REGION Network 4: Functional Test Station 6
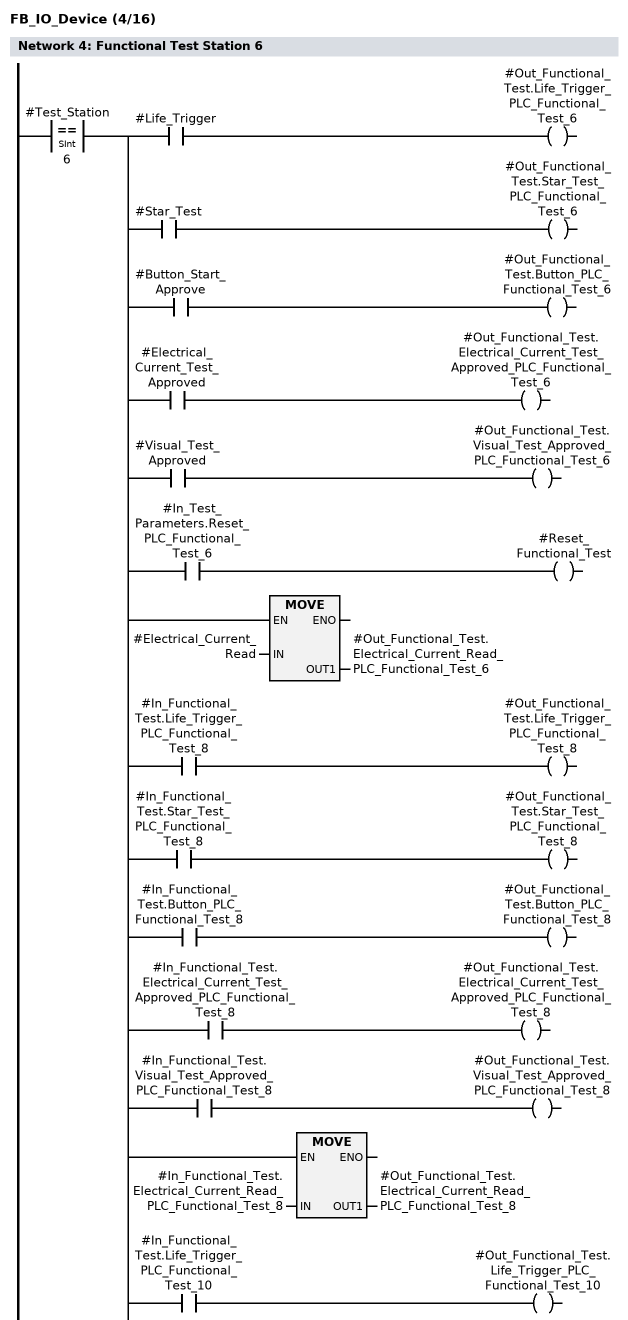
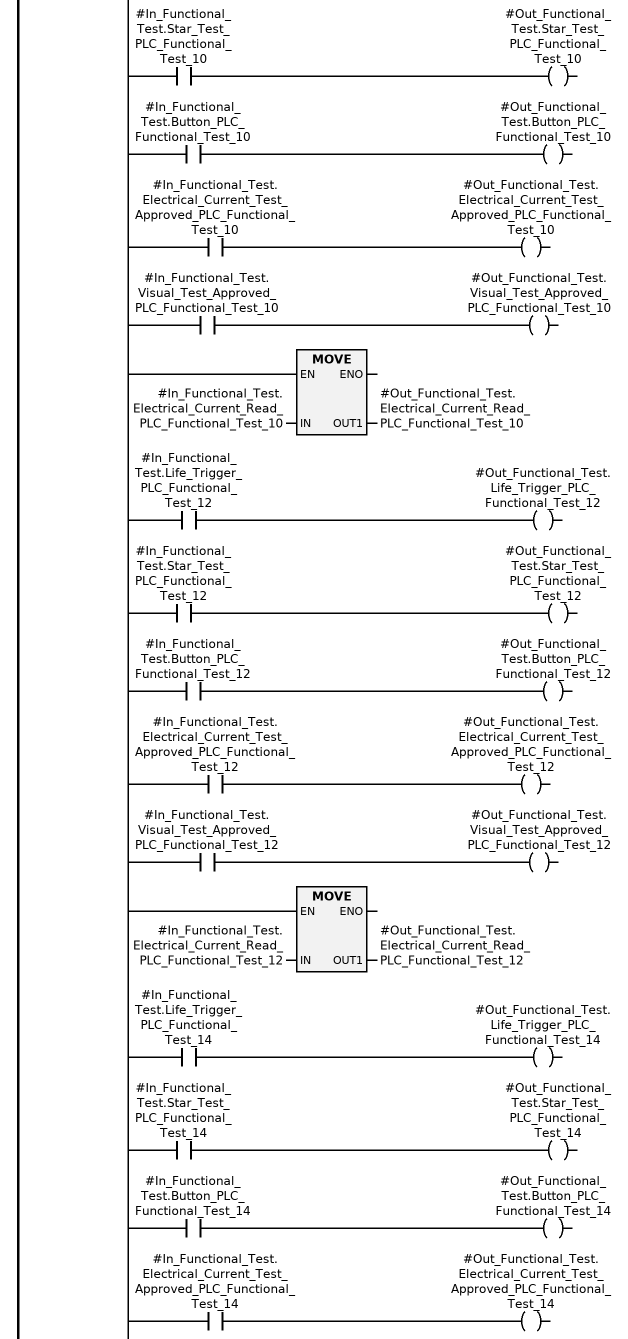
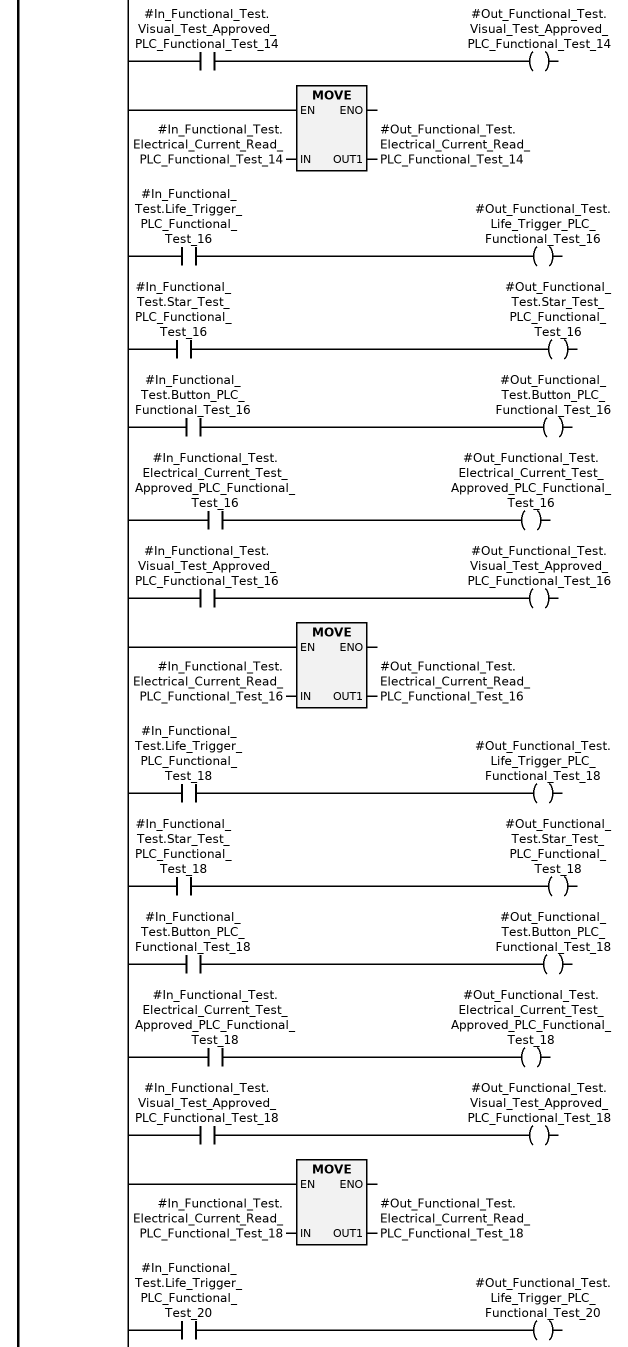
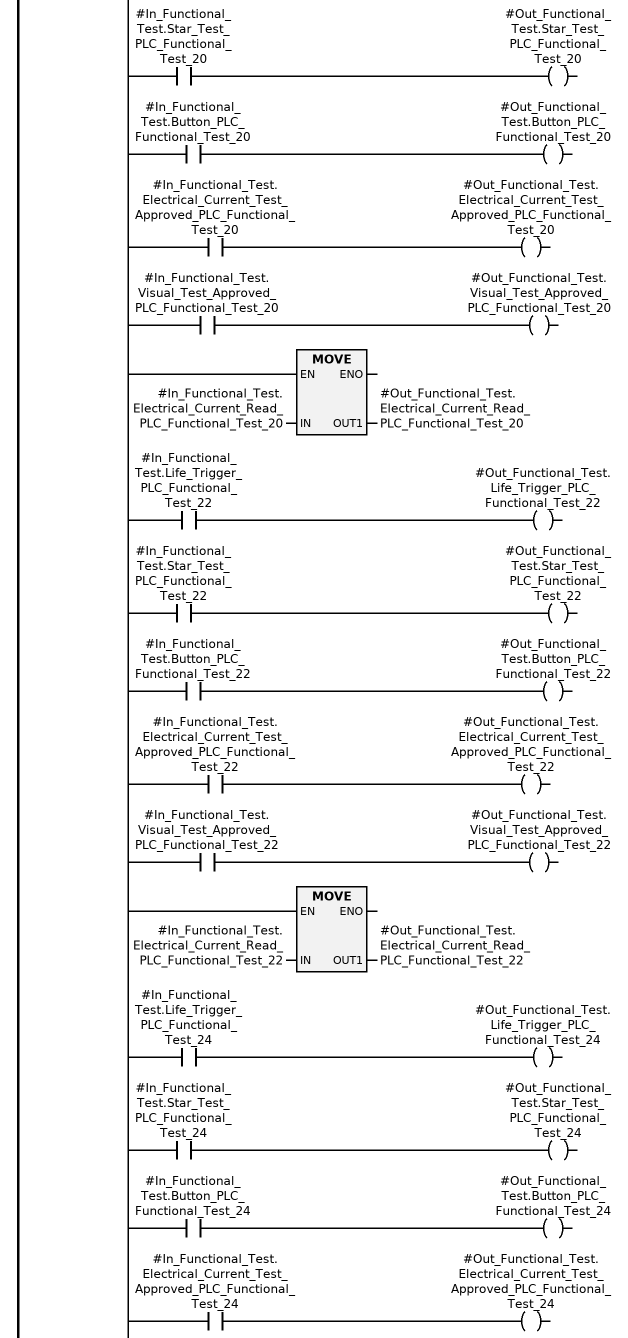
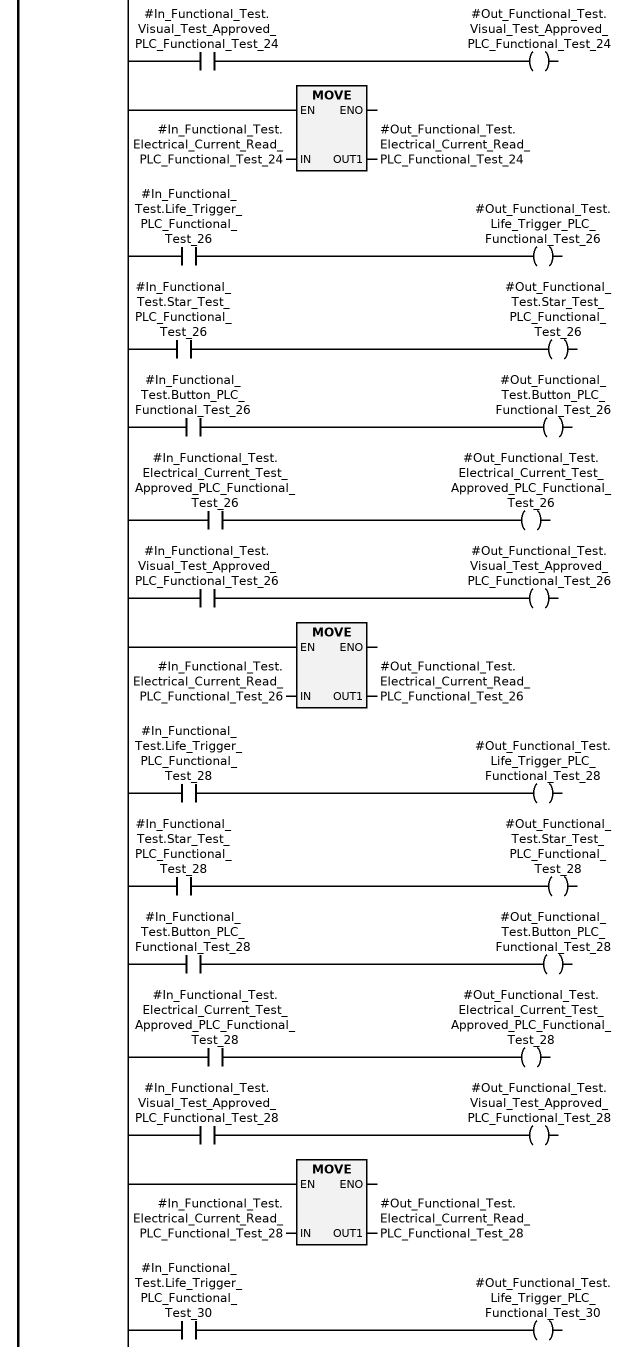
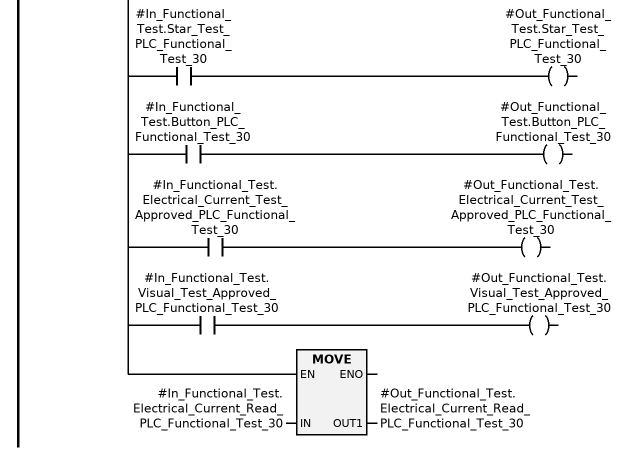
   RUNG wire#powerrail
      { S7_Templates := "SrcType := SInt" } EQ_Contact(in1 := #Test_Station, in2 := 6)
      wire#w1
      Contact( #Life_Trigger )
      Coil( #Out_Functional_Test.Life_Trigger_PLC_Functional_Test_6 )
   END_RUNG
   RUNG wire#w1
      Contact( #Star_Test )
      Coil( #Out_Functional_Test.Star_Test_PLC_Functional_Test_6 )
   END_RUNG
   RUNG wire#w1
      Contact( #Button_Start_Approve )
      Coil( #Out_Functional_Test.Button_PLC_Functional_Test_6 )
   END_RUNG
   RUNG wire#w1
      Contact( #Electrical_Current_Test_Approved )
      Coil( #Out_Functional_Test.Electrical_Current_Test_Approved_PLC_Functional_Test_6 )
   END_RUNG
   RUNG wire#w1
      Contact( #Visual_Test_Approved )
      Coil( #Out_Functional_Test.Visual_Test_Approved_PLC_Functional_Test_6 )
   END_RUNG
   RUNG wire#w1
      Contact( #In_Test_Parameters.Reset_PLC_Functional_Test_6 )
      Coil( #Reset_Functional_Test )
   END_RUNG
   RUNG wire#w1
      Move(in := #Electrical_Current_Read, out1 => #Out_Functional_Test.Electrical_Current_Read_PLC_Functional_Test_6)
   END_RUNG
   RUNG wire#w1
      Contact( #In_Functional_Test.Life_Trigger_PLC_Functional_Test_8 )
      Coil( #Out_Functional_Test.Life_Trigger_PLC_Functional_Test_8 )
   END_RUNG
   RUNG wire#w1
      Contact( #In_Functional_Test.Star_Test_PLC_Functional_Test_8 )
      Coil( #Out_Functional_Test.Star_Test_PLC_Functional_Test_8 )
   END_RUNG
   RUNG wire#w1
      Contact( #In_Functional_Test.Button_PLC_Functional_Test_8 )
      Coil( #Out_Functional_Test.Button_PLC_Functional_Test_8 )
   END_RUNG
   RUNG wire#w1
      Contact( #In_Functional_Test.Electrical_Current_Test_Approved_PLC_Functional_Test_8 )
      Coil( #Out_Functional_Test.Electrical_Current_Test_Approved_PLC_Functional_Test_8 )
   END_RUNG
   RUNG wire#w1
      Contact( #In_Functional_Test.Visual_Test_Approved_PLC_Functional_Test_8 )
      Coil( #Out_Functional_Test.Visual_Test_Approved_PLC_Functional_Test_8 )
   END_RUNG
   RUNG wire#w1
      Move(in := #In_Functional_Test.Electrical_Current_Read_PLC_Functional_Test_8, out1 => #Out_Functional_Test.Electrical_Current_Read_PLC_Functional_Test_8)
   END_RUNG
   RUNG wire#w1
      Contact( #In_Functional_Test.Life_Trigger_PLC_Functional_Test_10 )
      Coil( #Out_Functional_Test.Life_Trigger_PLC_Functional_Test_10 )
   END_RUNG
   RUNG wire#w1
      Contact( #In_Functional_Test.Star_Test_PLC_Functional_Test_10 )
      Coil( #Out_Functional_Test.Star_Test_PLC_Functional_Test_10 )
   END_RUNG
   RUNG wire#w1
      Contact( #In_Functional_Test.Button_PLC_Functional_Test_10 )
      Coil( #Out_Functional_Test.Button_PLC_Functional_Test_10 )
   END_RUNG
   RUNG wire#w1
      Contact( #In_Functional_Test.Electrical_Current_Test_Approved_PLC_Functional_Test_10 )
      Coil( #Out_Functional_Test.Electrical_Current_Test_Approved_PLC_Functional_Test_10 )
   END_RUNG
   RUNG wire#w1
      Contact( #In_Functional_Test.Visual_Test_Approved_PLC_Functional_Test_10 )
      Coil( #Out_Functional_Test.Visual_Test_Approved_PLC_Functional_Test_10 )
   END_RUNG
   RUNG wire#w1
      Move(in := #In_Functional_Test.Electrical_Current_Read_PLC_Functional_Test_10, out1 => #Out_Functional_Test.Electrical_Current_Read_PLC_Functional_Test_10)
   END_RUNG
   RUNG wire#w1
      Contact( #In_Functional_Test.Life_Trigger_PLC_Functional_Test_12 )
      Coil( #Out_Functional_Test.Life_Trigger_PLC_Functional_Test_12 )
   END_RUNG
   RUNG wire#w1
      Contact( #In_Functional_Test.Star_Test_PLC_Functional_Test_12 )
      Coil( #Out_Functional_Test.Star_Test_PLC_Functional_Test_12 )
   END_RUNG
   RUNG wire#w1
      Contact( #In_Functional_Test.Button_PLC_Functional_Test_12 )
      Coil( #Out_Functional_Test.Button_PLC_Functional_Test_12 )
   END_RUNG
   RUNG wire#w1
      Contact( #In_Functional_Test.Electrical_Current_Test_Approved_PLC_Functional_Test_12 )
      Coil( #Out_Functional_Test.Electrical_Current_Test_Approved_PLC_Functional_Test_12 )
   END_RUNG
   RUNG wire#w1
      Contact( #In_Functional_Test.Visual_Test_Approved_PLC_Functional_Test_12 )
      Coil( #Out_Functional_Test.Visual_Test_Approved_PLC_Functional_Test_12 )
   END_RUNG
   RUNG wire#w1
      Move(in := #In_Functional_Test.Electrical_Current_Read_PLC_Functional_Test_12, out1 => #Out_Functional_Test.Electrical_Current_Read_PLC_Functional_Test_12)
   END_RUNG
   RUNG wire#w1
      Contact( #In_Functional_Test.Life_Trigger_PLC_Functional_Test_14 )
      Coil( #Out_Functional_Test.Life_Trigger_PLC_Functional_Test_14 )
   END_RUNG
   RUNG wire#w1
      Contact( #In_Functional_Test.Star_Test_PLC_Functional_Test_14 )
      Coil( #Out_Functional_Test.Star_Test_PLC_Functional_Test_14 )
   END_RUNG
   RUNG wire#w1
      Contact( #In_Functional_Test.Button_PLC_Functional_Test_14 )
      Coil( #Out_Functional_Test.Button_PLC_Functional_Test_14 )
   END_RUNG
   RUNG wire#w1
      Contact( #In_Functional_Test.Electrical_Current_Test_Approved_PLC_Functional_Test_14 )
      Coil( #Out_Functional_Test.Electrical_Current_Test_Approved_PLC_Functional_Test_14 )
   END_RUNG
   RUNG wire#w1
      Contact( #In_Functional_Test.Visual_Test_Approved_PLC_Functional_Test_14 )
      Coil( #Out_Functional_Test.Visual_Test_Approved_PLC_Functional_Test_14 )
   END_RUNG
   RUNG wire#w1
      Move(in := #In_Functional_Test.Electrical_Current_Read_PLC_Functional_Test_14, out1 => #Out_Functional_Test.Electrical_Current_Read_PLC_Functional_Test_14)
   END_RUNG
   RUNG wire#w1
      Contact( #In_Functional_Test.Life_Trigger_PLC_Functional_Test_16 )
      Coil( #Out_Functional_Test.Life_Trigger_PLC_Functional_Test_16 )
   END_RUNG
   RUNG wire#w1
      Contact( #In_Functional_Test.Star_Test_PLC_Functional_Test_16 )
      Coil( #Out_Functional_Test.Star_Test_PLC_Functional_Test_16 )
   END_RUNG
   RUNG wire#w1
      Contact( #In_Functional_Test.Button_PLC_Functional_Test_16 )
      Coil( #Out_Functional_Test.Button_PLC_Functional_Test_16 )
   END_RUNG
   RUNG wire#w1
      Contact( #In_Functional_Test.Electrical_Current_Test_Approved_PLC_Functional_Test_16 )
      Coil( #Out_Functional_Test.Electrical_Current_Test_Approved_PLC_Functional_Test_16 )
   END_RUNG
   RUNG wire#w1
      Contact( #In_Functional_Test.Visual_Test_Approved_PLC_Functional_Test_16 )
      Coil( #Out_Functional_Test.Visual_Test_Approved_PLC_Functional_Test_16 )
   END_RUNG
   RUNG wire#w1
      Move(in := #In_Functional_Test.Electrical_Current_Read_PLC_Functional_Test_16, out1 => #Out_Functional_Test.Electrical_Current_Read_PLC_Functional_Test_16)
   END_RUNG
   RUNG wire#w1
      Contact( #In_Functional_Test.Life_Trigger_PLC_Functional_Test_18 )
      Coil( #Out_Functional_Test.Life_Trigger_PLC_Functional_Test_18 )
   END_RUNG
   RUNG wire#w1
      Contact( #In_Functional_Test.Star_Test_PLC_Functional_Test_18 )
      Coil( #Out_Functional_Test.Star_Test_PLC_Functional_Test_18 )
   END_RUNG
   RUNG wire#w1
      Contact( #In_Functional_Test.Button_PLC_Functional_Test_18 )
      Coil( #Out_Functional_Test.Button_PLC_Functional_Test_18 )
   END_RUNG
   RUNG wire#w1
      Contact( #In_Functional_Test.Electrical_Current_Test_Approved_PLC_Functional_Test_18 )
      Coil( #Out_Functional_Test.Electrical_Current_Test_Approved_PLC_Functional_Test_18 )
   END_RUNG
   RUNG wire#w1
      Contact( #In_Functional_Test.Visual_Test_Approved_PLC_Functional_Test_18 )
      Coil( #Out_Functional_Test.Visual_Test_Approved_PLC_Functional_Test_18 )
   END_RUNG
   RUNG wire#w1
      Move(in := #In_Functional_Test.Electrical_Current_Read_PLC_Functional_Test_18, out1 => #Out_Functional_Test.Electrical_Current_Read_PLC_Functional_Test_18)
   END_RUNG
   RUNG wire#w1
      Contact( #In_Functional_Test.Life_Trigger_PLC_Functional_Test_20 )
      Coil( #Out_Functional_Test.Life_Trigger_PLC_Functional_Test_20 )
   END_RUNG
   RUNG wire#w1
      Contact( #In_Functional_Test.Star_Test_PLC_Functional_Test_20 )
      Coil( #Out_Functional_Test.Star_Test_PLC_Functional_Test_20 )
   END_RUNG
   RUNG wire#w1
      Contact( #In_Functional_Test.Button_PLC_Functional_Test_20 )
      Coil( #Out_Functional_Test.Button_PLC_Functional_Test_20 )
   END_RUNG
   RUNG wire#w1
      Contact( #In_Functional_Test.Electrical_Current_Test_Approved_PLC_Functional_Test_20 )
      Coil( #Out_Functional_Test.Electrical_Current_Test_Approved_PLC_Functional_Test_20 )
   END_RUNG
   RUNG wire#w1
      Contact( #In_Functional_Test.Visual_Test_Approved_PLC_Functional_Test_20 )
      Coil( #Out_Functional_Test.Visual_Test_Approved_PLC_Functional_Test_20 )
   END_RUNG
   RUNG wire#w1
      Move(in := #In_Functional_Test.Electrical_Current_Read_PLC_Functional_Test_20, out1 => #Out_Functional_Test.Electrical_Current_Read_PLC_Functional_Test_20)
   END_RUNG
   RUNG wire#w1
      Contact( #In_Functional_Test.Life_Trigger_PLC_Functional_Test_22 )
      Coil( #Out_Functional_Test.Life_Trigger_PLC_Functional_Test_22 )
   END_RUNG
   RUNG wire#w1
      Contact( #In_Functional_Test.Star_Test_PLC_Functional_Test_22 )
      Coil( #Out_Functional_Test.Star_Test_PLC_Functional_Test_22 )
   END_RUNG
   RUNG wire#w1
      Contact( #In_Functional_Test.Button_PLC_Functional_Test_22 )
      Coil( #Out_Functional_Test.Button_PLC_Functional_Test_22 )
   END_RUNG
   RUNG wire#w1
      Contact( #In_Functional_Test.Electrical_Current_Test_Approved_PLC_Functional_Test_22 )
      Coil( #Out_Functional_Test.Electrical_Current_Test_Approved_PLC_Functional_Test_22 )
   END_RUNG
   RUNG wire#w1
      Contact( #In_Functional_Test.Visual_Test_Approved_PLC_Functional_Test_22 )
      Coil( #Out_Functional_Test.Visual_Test_Approved_PLC_Functional_Test_22 )
   END_RUNG
   RUNG wire#w1
      Move(in := #In_Functional_Test.Electrical_Current_Read_PLC_Functional_Test_22, out1 => #Out_Functional_Test.Electrical_Current_Read_PLC_Functional_Test_22)
   END_RUNG
   RUNG wire#w1
      Contact( #In_Functional_Test.Life_Trigger_PLC_Functional_Test_24 )
      Coil( #Out_Functional_Test.Life_Trigger_PLC_Functional_Test_24 )
   END_RUNG
   RUNG wire#w1
      Contact( #In_Functional_Test.Star_Test_PLC_Functional_Test_24 )
      Coil( #Out_Functional_Test.Star_Test_PLC_Functional_Test_24 )
   END_RUNG
   RUNG wire#w1
      Contact( #In_Functional_Test.Button_PLC_Functional_Test_24 )
      Coil( #Out_Functional_Test.Button_PLC_Functional_Test_24 )
   END_RUNG
   RUNG wire#w1
      Contact( #In_Functional_Test.Electrical_Current_Test_Approved_PLC_Functional_Test_24 )
      Coil( #Out_Functional_Test.Electrical_Current_Test_Approved_PLC_Functional_Test_24 )
   END_RUNG
   RUNG wire#w1
      Contact( #In_Functional_Test.Visual_Test_Approved_PLC_Functional_Test_24 )
      Coil( #Out_Functional_Test.Visual_Test_Approved_PLC_Functional_Test_24 )
   END_RUNG
   RUNG wire#w1
      Move(in := #In_Functional_Test.Electrical_Current_Read_PLC_Functional_Test_24, out1 => #Out_Functional_Test.Electrical_Current_Read_PLC_Functional_Test_24)
   END_RUNG
   RUNG wire#w1
      Contact( #In_Functional_Test.Life_Trigger_PLC_Functional_Test_26 )
      Coil( #Out_Functional_Test.Life_Trigger_PLC_Functional_Test_26 )
   END_RUNG
   RUNG wire#w1
      Contact( #In_Functional_Test.Star_Test_PLC_Functional_Test_26 )
      Coil( #Out_Functional_Test.Star_Test_PLC_Functional_Test_26 )
   END_RUNG
   RUNG wire#w1
      Contact( #In_Functional_Test.Button_PLC_Functional_Test_26 )
      Coil( #Out_Functional_Test.Button_PLC_Functional_Test_26 )
   END_RUNG
   RUNG wire#w1
      Contact( #In_Functional_Test.Electrical_Current_Test_Approved_PLC_Functional_Test_26 )
      Coil( #Out_Functional_Test.Electrical_Current_Test_Approved_PLC_Functional_Test_26 )
   END_RUNG
   RUNG wire#w1
      Contact( #In_Functional_Test.Visual_Test_Approved_PLC_Functional_Test_26 )
      Coil( #Out_Functional_Test.Visual_Test_Approved_PLC_Functional_Test_26 )
   END_RUNG
   RUNG wire#w1
      Move(in := #In_Functional_Test.Electrical_Current_Read_PLC_Functional_Test_26, out1 => #Out_Functional_Test.Electrical_Current_Read_PLC_Functional_Test_26)
   END_RUNG
   RUNG wire#w1
      Contact( #In_Functional_Test.Life_Trigger_PLC_Functional_Test_28 )
      Coil( #Out_Functional_Test.Life_Trigger_PLC_Functional_Test_28 )
   END_RUNG
   RUNG wire#w1
      Contact( #In_Functional_Test.Star_Test_PLC_Functional_Test_28 )
      Coil( #Out_Functional_Test.Star_Test_PLC_Functional_Test_28 )
   END_RUNG
   RUNG wire#w1
      Contact( #In_Functional_Test.Button_PLC_Functional_Test_28 )
      Coil( #Out_Functional_Test.Button_PLC_Functional_Test_28 )
   END_RUNG
   RUNG wire#w1
      Contact( #In_Functional_Test.Electrical_Current_Test_Approved_PLC_Functional_Test_28 )
      Coil( #Out_Functional_Test.Electrical_Current_Test_Approved_PLC_Functional_Test_28 )
   END_RUNG
   RUNG wire#w1
      Contact( #In_Functional_Test.Visual_Test_Approved_PLC_Functional_Test_28 )
      Coil( #Out_Functional_Test.Visual_Test_Approved_PLC_Functional_Test_28 )
   END_RUNG
   RUNG wire#w1
      Move(in := #In_Functional_Test.Electrical_Current_Read_PLC_Functional_Test_28, out1 => #Out_Functional_Test.Electrical_Current_Read_PLC_Functional_Test_28)
   END_RUNG
   RUNG wire#w1
      Contact( #In_Functional_Test.Life_Trigger_PLC_Functional_Test_30 )
      Coil( #Out_Functional_Test.Life_Trigger_PLC_Functional_Test_30 )
   END_RUNG
   RUNG wire#w1
      Contact( #In_Functional_Test.Star_Test_PLC_Functional_Test_30 )
      Coil( #Out_Functional_Test.Star_Test_PLC_Functional_Test_30 )
   END_RUNG
   RUNG wire#w1
      Contact( #In_Functional_Test.Button_PLC_Functional_Test_30 )
      Coil( #Out_Functional_Test.Button_PLC_Functional_Test_30 )
   END_RUNG
   RUNG wire#w1
      Contact( #In_Functional_Test.Electrical_Current_Test_Approved_PLC_Functional_Test_30 )
      Coil( #Out_Functional_Test.Electrical_Current_Test_Approved_PLC_Functional_Test_30 )
   END_RUNG
   RUNG wire#w1
      Contact( #In_Functional_Test.Visual_Test_Approved_PLC_Functional_Test_30 )
      Coil( #Out_Functional_Test.Visual_Test_Approved_PLC_Functional_Test_30 )
   END_RUNG
   RUNG wire#w1
      Move(in := #In_Functional_Test.Electrical_Current_Read_PLC_Functional_Test_30, out1 => #Out_Functional_Test.Electrical_Current_Read_PLC_Functional_Test_30)
   END_RUNG
   // the same network as SCL:
   #_w1 := #Test_Station = 6;
   #Out_Functional_Test.Life_Trigger_PLC_Functional_Test_6 := #_w1 AND #Life_Trigger;
   #Out_Functional_Test.Star_Test_PLC_Functional_Test_6 := #_w1 AND #Star_Test;
   #Out_Functional_Test.Button_PLC_Functional_Test_6 := #_w1 AND #Button_Start_Approve;
   #Out_Functional_Test.Electrical_Current_Test_Approved_PLC_Functional_Test_6 := #_w1 AND #Electrical_Current_Test_Approved;
   #Out_Functional_Test.Visual_Test_Approved_PLC_Functional_Test_6 := #_w1 AND #Visual_Test_Approved;
   #Reset_Functional_Test := #_w1 AND #In_Test_Parameters.Reset_PLC_Functional_Test_6;
   IF #_w1 THEN
       #Out_Functional_Test.Electrical_Current_Read_PLC_Functional_Test_6 := #Electrical_Current_Read;
   END_IF;
   #Out_Functional_Test.Life_Trigger_PLC_Functional_Test_8 := #_w1 AND #In_Functional_Test.Life_Trigger_PLC_Functional_Test_8;
   #Out_Functional_Test.Star_Test_PLC_Functional_Test_8 := #_w1 AND #In_Functional_Test.Star_Test_PLC_Functional_Test_8;
   #Out_Functional_Test.Button_PLC_Functional_Test_8 := #_w1 AND #In_Functional_Test.Button_PLC_Functional_Test_8;
   #Out_Functional_Test.Electrical_Current_Test_Approved_PLC_Functional_Test_8 := #_w1 AND #In_Functional_Test.Electrical_Current_Test_Approved_PLC_Functional_Test_8;
   #Out_Functional_Test.Visual_Test_Approved_PLC_Functional_Test_8 := #_w1 AND #In_Functional_Test.Visual_Test_Approved_PLC_Functional_Test_8;
   IF #_w1 THEN
       #Out_Functional_Test.Electrical_Current_Read_PLC_Functional_Test_8 := #In_Functional_Test.Electrical_Current_Read_PLC_Functional_Test_8;
   END_IF;
   #Out_Functional_Test.Life_Trigger_PLC_Functional_Test_10 := #_w1 AND #In_Functional_Test.Life_Trigger_PLC_Functional_Test_10;
   #Out_Functional_Test.Star_Test_PLC_Functional_Test_10 := #_w1 AND #In_Functional_Test.Star_Test_PLC_Functional_Test_10;
   #Out_Functional_Test.Button_PLC_Functional_Test_10 := #_w1 AND #In_Functional_Test.Button_PLC_Functional_Test_10;
   #Out_Functional_Test.Electrical_Current_Test_Approved_PLC_Functional_Test_10 := #_w1 AND #In_Functional_Test.Electrical_Current_Test_Approved_PLC_Functional_Test_10;
   #Out_Functional_Test.Visual_Test_Approved_PLC_Functional_Test_10 := #_w1 AND #In_Functional_Test.Visual_Test_Approved_PLC_Functional_Test_10;
   IF #_w1 THEN
       #Out_Functional_Test.Electrical_Current_Read_PLC_Functional_Test_10 := #In_Functional_Test.Electrical_Current_Read_PLC_Functional_Test_10;
   END_IF;
   #Out_Functional_Test.Life_Trigger_PLC_Functional_Test_12 := #_w1 AND #In_Functional_Test.Life_Trigger_PLC_Functional_Test_12;
   #Out_Functional_Test.Star_Test_PLC_Functional_Test_12 := #_w1 AND #In_Functional_Test.Star_Test_PLC_Functional_Test_12;
   #Out_Functional_Test.Button_PLC_Functional_Test_12 := #_w1 AND #In_Functional_Test.Button_PLC_Functional_Test_12;
   #Out_Functional_Test.Electrical_Current_Test_Approved_PLC_Functional_Test_12 := #_w1 AND #In_Functional_Test.Electrical_Current_Test_Approved_PLC_Functional_Test_12;
   #Out_Functional_Test.Visual_Test_Approved_PLC_Functional_Test_12 := #_w1 AND #In_Functional_Test.Visual_Test_Approved_PLC_Functional_Test_12;
   IF #_w1 THEN
       #Out_Functional_Test.Electrical_Current_Read_PLC_Functional_Test_12 := #In_Functional_Test.Electrical_Current_Read_PLC_Functional_Test_12;
   END_IF;
   #Out_Functional_Test.Life_Trigger_PLC_Functional_Test_14 := #_w1 AND #In_Functional_Test.Life_Trigger_PLC_Functional_Test_14;
   #Out_Functional_Test.Star_Test_PLC_Functional_Test_14 := #_w1 AND #In_Functional_Test.Star_Test_PLC_Functional_Test_14;
   #Out_Functional_Test.Button_PLC_Functional_Test_14 := #_w1 AND #In_Functional_Test.Button_PLC_Functional_Test_14;
   #Out_Functional_Test.Electrical_Current_Test_Approved_PLC_Functional_Test_14 := #_w1 AND #In_Functional_Test.Electrical_Current_Test_Approved_PLC_Functional_Test_14;
   #Out_Functional_Test.Visual_Test_Approved_PLC_Functional_Test_14 := #_w1 AND #In_Functional_Test.Visual_Test_Approved_PLC_Functional_Test_14;
   IF #_w1 THEN
       #Out_Functional_Test.Electrical_Current_Read_PLC_Functional_Test_14 := #In_Functional_Test.Electrical_Current_Read_PLC_Functional_Test_14;
   END_IF;
   #Out_Functional_Test.Life_Trigger_PLC_Functional_Test_16 := #_w1 AND #In_Functional_Test.Life_Trigger_PLC_Functional_Test_16;
   #Out_Functional_Test.Star_Test_PLC_Functional_Test_16 := #_w1 AND #In_Functional_Test.Star_Test_PLC_Functional_Test_16;
   #Out_Functional_Test.Button_PLC_Functional_Test_16 := #_w1 AND #In_Functional_Test.Button_PLC_Functional_Test_16;
   #Out_Functional_Test.Electrical_Current_Test_Approved_PLC_Functional_Test_16 := #_w1 AND #In_Functional_Test.Electrical_Current_Test_Approved_PLC_Functional_Test_16;
   #Out_Functional_Test.Visual_Test_Approved_PLC_Functional_Test_16 := #_w1 AND #In_Functional_Test.Visual_Test_Approved_PLC_Functional_Test_16;
   IF #_w1 THEN
       #Out_Functional_Test.Electrical_Current_Read_PLC_Functional_Test_16 := #In_Functional_Test.Electrical_Current_Read_PLC_Functional_Test_16;
   END_IF;
   #Out_Functional_Test.Life_Trigger_PLC_Functional_Test_18 := #_w1 AND #In_Functional_Test.Life_Trigger_PLC_Functional_Test_18;
   #Out_Functional_Test.Star_Test_PLC_Functional_Test_18 := #_w1 AND #In_Functional_Test.Star_Test_PLC_Functional_Test_18;
   #Out_Functional_Test.Button_PLC_Functional_Test_18 := #_w1 AND #In_Functional_Test.Button_PLC_Functional_Test_18;
   #Out_Functional_Test.Electrical_Current_Test_Approved_PLC_Functional_Test_18 := #_w1 AND #In_Functional_Test.Electrical_Current_Test_Approved_PLC_Functional_Test_18;
   #Out_Functional_Test.Visual_Test_Approved_PLC_Functional_Test_18 := #_w1 AND #In_Functional_Test.Visual_Test_Approved_PLC_Functional_Test_18;
   IF #_w1 THEN
       #Out_Functional_Test.Electrical_Current_Read_PLC_Functional_Test_18 := #In_Functional_Test.Electrical_Current_Read_PLC_Functional_Test_18;
   END_IF;
   #Out_Functional_Test.Life_Trigger_PLC_Functional_Test_20 := #_w1 AND #In_Functional_Test.Life_Trigger_PLC_Functional_Test_20;
   #Out_Functional_Test.Star_Test_PLC_Functional_Test_20 := #_w1 AND #In_Functional_Test.Star_Test_PLC_Functional_Test_20;
   #Out_Functional_Test.Button_PLC_Functional_Test_20 := #_w1 AND #In_Functional_Test.Button_PLC_Functional_Test_20;
   #Out_Functional_Test.Electrical_Current_Test_Approved_PLC_Functional_Test_20 := #_w1 AND #In_Functional_Test.Electrical_Current_Test_Approved_PLC_Functional_Test_20;
   #Out_Functional_Test.Visual_Test_Approved_PLC_Functional_Test_20 := #_w1 AND #In_Functional_Test.Visual_Test_Approved_PLC_Functional_Test_20;
   IF #_w1 THEN
       #Out_Functional_Test.Electrical_Current_Read_PLC_Functional_Test_20 := #In_Functional_Test.Electrical_Current_Read_PLC_Functional_Test_20;
   END_IF;
   #Out_Functional_Test.Life_Trigger_PLC_Functional_Test_22 := #_w1 AND #In_Functional_Test.Life_Trigger_PLC_Functional_Test_22;
   #Out_Functional_Test.Star_Test_PLC_Functional_Test_22 := #_w1 AND #In_Functional_Test.Star_Test_PLC_Functional_Test_22;
   #Out_Functional_Test.Button_PLC_Functional_Test_22 := #_w1 AND #In_Functional_Test.Button_PLC_Functional_Test_22;
   #Out_Functional_Test.Electrical_Current_Test_Approved_PLC_Functional_Test_22 := #_w1 AND #In_Functional_Test.Electrical_Current_Test_Approved_PLC_Functional_Test_22;
   #Out_Functional_Test.Visual_Test_Approved_PLC_Functional_Test_22 := #_w1 AND #In_Functional_Test.Visual_Test_Approved_PLC_Functional_Test_22;
   IF #_w1 THEN
       #Out_Functional_Test.Electrical_Current_Read_PLC_Functional_Test_22 := #In_Functional_Test.Electrical_Current_Read_PLC_Functional_Test_22;
   END_IF;
   #Out_Functional_Test.Life_Trigger_PLC_Functional_Test_24 := #_w1 AND #In_Functional_Test.Life_Trigger_PLC_Functional_Test_24;
   #Out_Functional_Test.Star_Test_PLC_Functional_Test_24 := #_w1 AND #In_Functional_Test.Star_Test_PLC_Functional_Test_24;
   #Out_Functional_Test.Button_PLC_Functional_Test_24 := #_w1 AND #In_Functional_Test.Button_PLC_Functional_Test_24;
   #Out_Functional_Test.Electrical_Current_Test_Approved_PLC_Functional_Test_24 := #_w1 AND #In_Functional_Test.Electrical_Current_Test_Approved_PLC_Functional_Test_24;
   #Out_Functional_Test.Visual_Test_Approved_PLC_Functional_Test_24 := #_w1 AND #In_Functional_Test.Visual_Test_Approved_PLC_Functional_Test_24;
   IF #_w1 THEN
       #Out_Functional_Test.Electrical_Current_Read_PLC_Functional_Test_24 := #In_Functional_Test.Electrical_Current_Read_PLC_Functional_Test_24;
   END_IF;
   #Out_Functional_Test.Life_Trigger_PLC_Functional_Test_26 := #_w1 AND #In_Functional_Test.Life_Trigger_PLC_Functional_Test_26;
   #Out_Functional_Test.Star_Test_PLC_Functional_Test_26 := #_w1 AND #In_Functional_Test.Star_Test_PLC_Functional_Test_26;
   #Out_Functional_Test.Button_PLC_Functional_Test_26 := #_w1 AND #In_Functional_Test.Button_PLC_Functional_Test_26;
   #Out_Functional_Test.Electrical_Current_Test_Approved_PLC_Functional_Test_26 := #_w1 AND #In_Functional_Test.Electrical_Current_Test_Approved_PLC_Functional_Test_26;
   #Out_Functional_Test.Visual_Test_Approved_PLC_Functional_Test_26 := #_w1 AND #In_Functional_Test.Visual_Test_Approved_PLC_Functional_Test_26;
   IF #_w1 THEN
       #Out_Functional_Test.Electrical_Current_Read_PLC_Functional_Test_26 := #In_Functional_Test.Electrical_Current_Read_PLC_Functional_Test_26;
   END_IF;
   #Out_Functional_Test.Life_Trigger_PLC_Functional_Test_28 := #_w1 AND #In_Functional_Test.Life_Trigger_PLC_Functional_Test_28;
   #Out_Functional_Test.Star_Test_PLC_Functional_Test_28 := #_w1 AND #In_Functional_Test.Star_Test_PLC_Functional_Test_28;
   #Out_Functional_Test.Button_PLC_Functional_Test_28 := #_w1 AND #In_Functional_Test.Button_PLC_Functional_Test_28;
   #Out_Functional_Test.Electrical_Current_Test_Approved_PLC_Functional_Test_28 := #_w1 AND #In_Functional_Test.Electrical_Current_Test_Approved_PLC_Functional_Test_28;
   #Out_Functional_Test.Visual_Test_Approved_PLC_Functional_Test_28 := #_w1 AND #In_Functional_Test.Visual_Test_Approved_PLC_Functional_Test_28;
   IF #_w1 THEN
       #Out_Functional_Test.Electrical_Current_Read_PLC_Functional_Test_28 := #In_Functional_Test.Electrical_Current_Read_PLC_Functional_Test_28;
   END_IF;
   #Out_Functional_Test.Life_Trigger_PLC_Functional_Test_30 := #_w1 AND #In_Functional_Test.Life_Trigger_PLC_Functional_Test_30;
   #Out_Functional_Test.Star_Test_PLC_Functional_Test_30 := #_w1 AND #In_Functional_Test.Star_Test_PLC_Functional_Test_30;
   #Out_Functional_Test.Button_PLC_Functional_Test_30 := #_w1 AND #In_Functional_Test.Button_PLC_Functional_Test_30;
   #Out_Functional_Test.Electrical_Current_Test_Approved_PLC_Functional_Test_30 := #_w1 AND #In_Functional_Test.Electrical_Current_Test_Approved_PLC_Functional_Test_30;
   #Out_Functional_Test.Visual_Test_Approved_PLC_Functional_Test_30 := #_w1 AND #In_Functional_Test.Visual_Test_Approved_PLC_Functional_Test_30;
   IF #_w1 THEN
       #Out_Functional_Test.Electrical_Current_Read_PLC_Functional_Test_30 := #In_Functional_Test.Electrical_Current_Read_PLC_Functional_Test_30;
   END_IF;
END_REGION

REGION Network 5: Functional Test Station 8
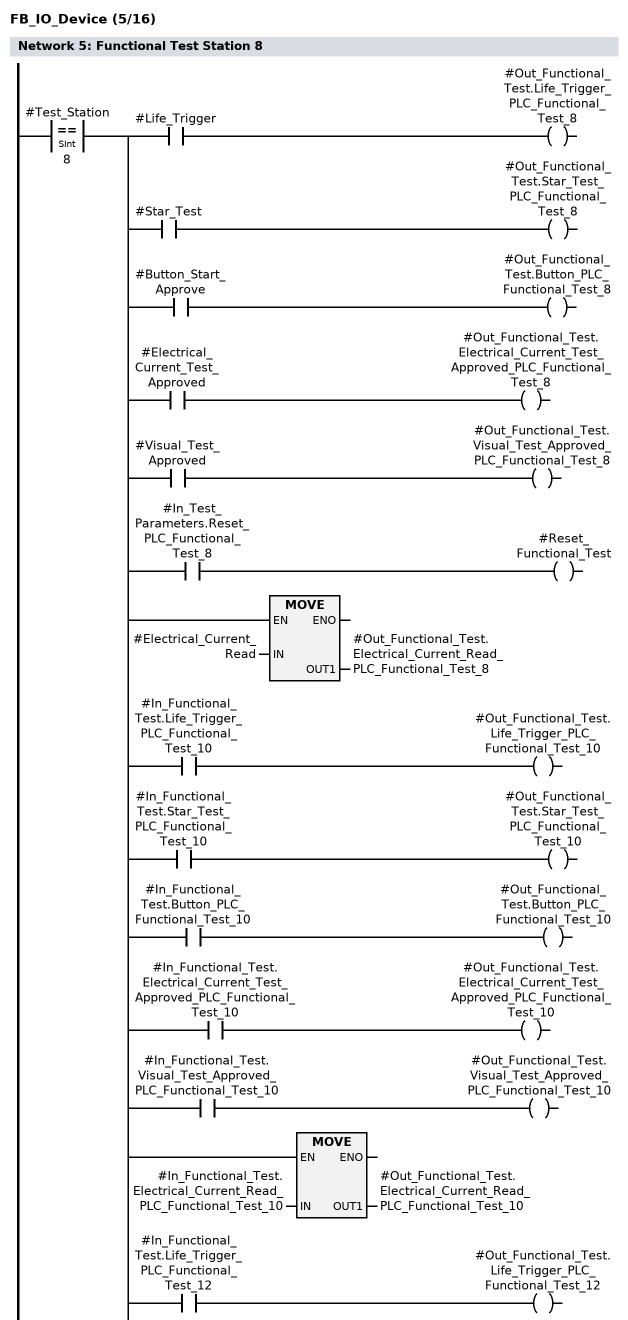
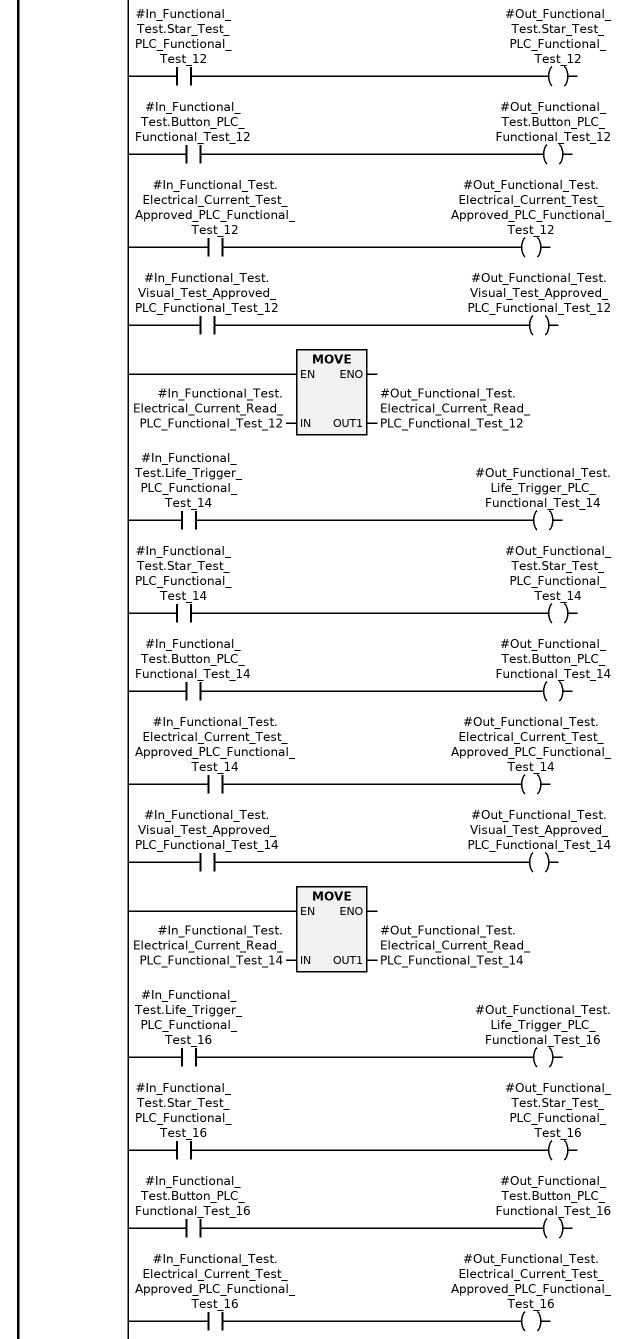
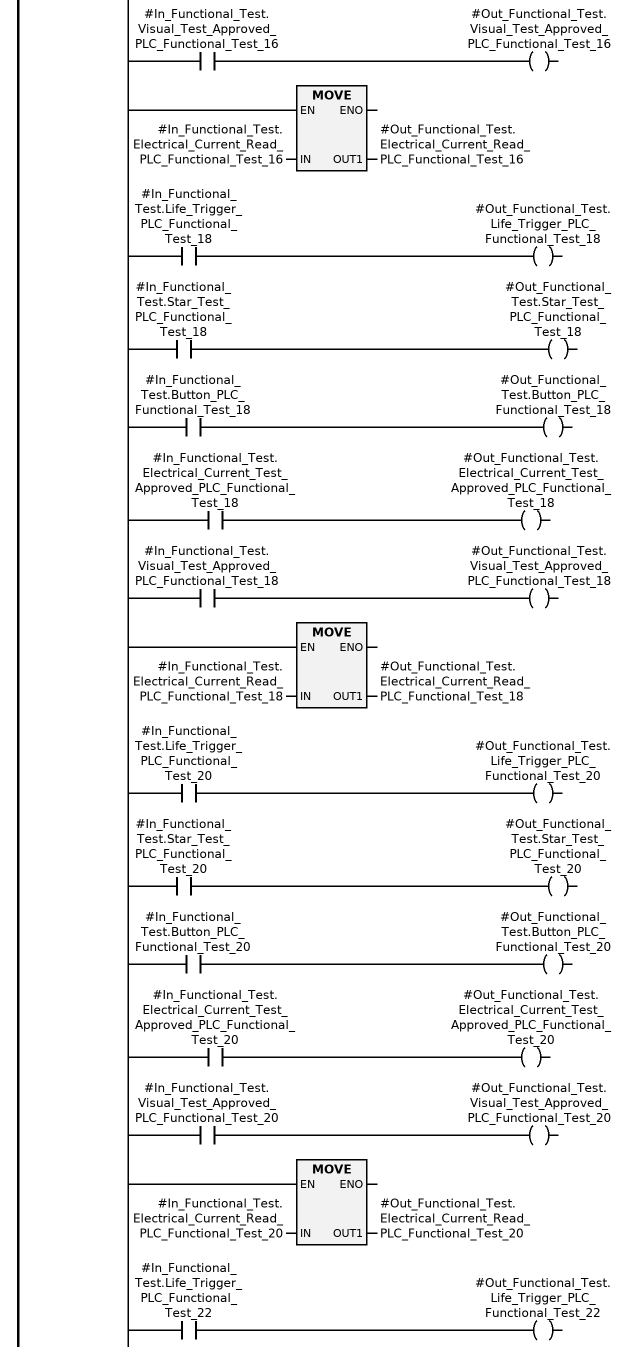
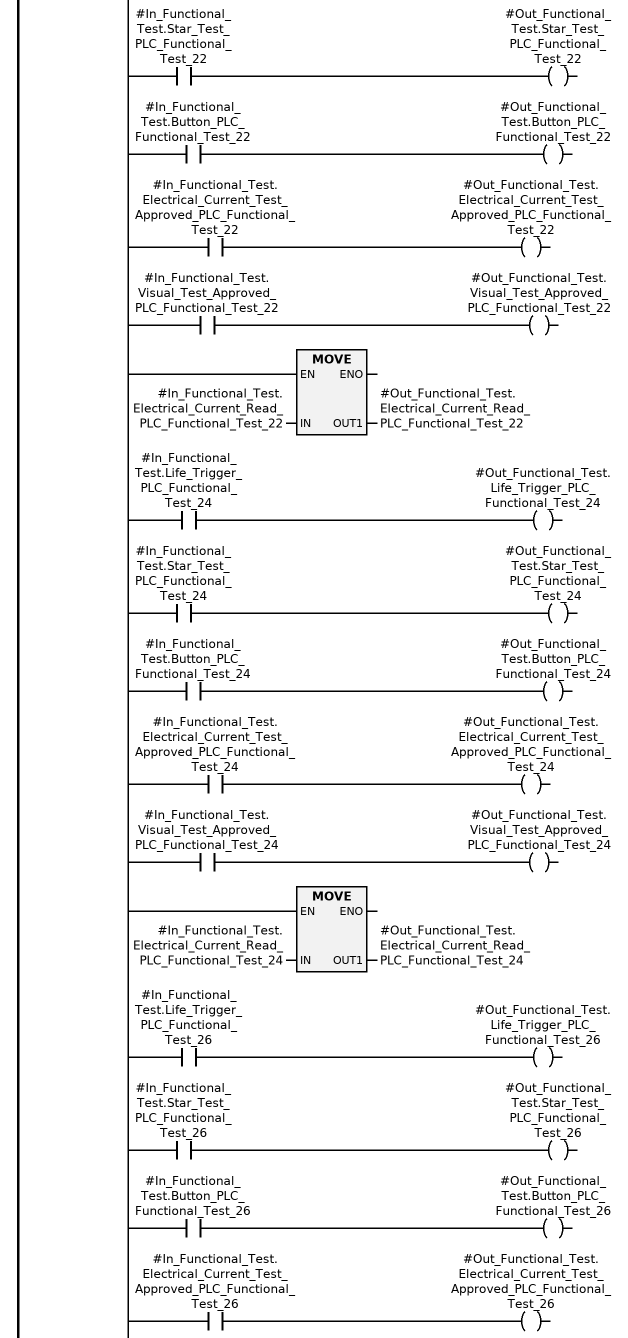
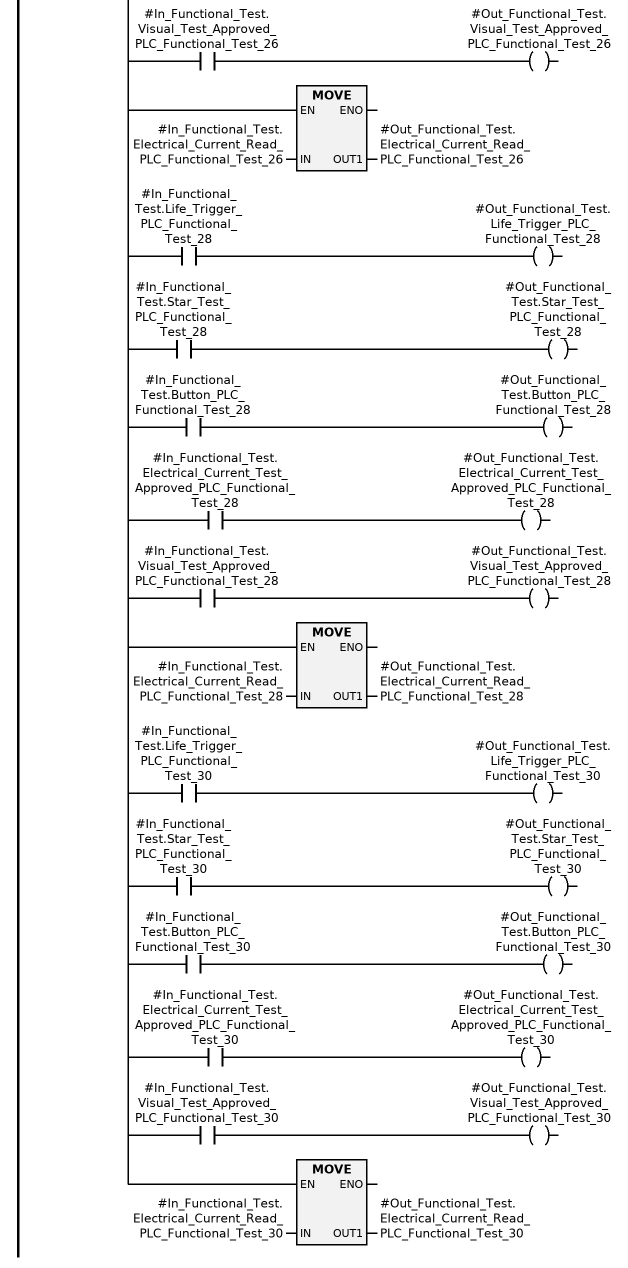
   RUNG wire#powerrail
      { S7_Templates := "SrcType := SInt" } EQ_Contact(in1 := #Test_Station, in2 := 8)
      wire#w1
      Contact( #Life_Trigger )
      Coil( #Out_Functional_Test.Life_Trigger_PLC_Functional_Test_8 )
   END_RUNG
   RUNG wire#w1
      Contact( #Star_Test )
      Coil( #Out_Functional_Test.Star_Test_PLC_Functional_Test_8 )
   END_RUNG
   RUNG wire#w1
      Contact( #Button_Start_Approve )
      Coil( #Out_Functional_Test.Button_PLC_Functional_Test_8 )
   END_RUNG
   RUNG wire#w1
      Contact( #Electrical_Current_Test_Approved )
      Coil( #Out_Functional_Test.Electrical_Current_Test_Approved_PLC_Functional_Test_8 )
   END_RUNG
   RUNG wire#w1
      Contact( #Visual_Test_Approved )
      Coil( #Out_Functional_Test.Visual_Test_Approved_PLC_Functional_Test_8 )
   END_RUNG
   RUNG wire#w1
      Contact( #In_Test_Parameters.Reset_PLC_Functional_Test_8 )
      Coil( #Reset_Functional_Test )
   END_RUNG
   RUNG wire#w1
      Move(in := #Electrical_Current_Read, out1 => #Out_Functional_Test.Electrical_Current_Read_PLC_Functional_Test_8)
   END_RUNG
   RUNG wire#w1
      Contact( #In_Functional_Test.Life_Trigger_PLC_Functional_Test_10 )
      Coil( #Out_Functional_Test.Life_Trigger_PLC_Functional_Test_10 )
   END_RUNG
   RUNG wire#w1
      Contact( #In_Functional_Test.Star_Test_PLC_Functional_Test_10 )
      Coil( #Out_Functional_Test.Star_Test_PLC_Functional_Test_10 )
   END_RUNG
   RUNG wire#w1
      Contact( #In_Functional_Test.Button_PLC_Functional_Test_10 )
      Coil( #Out_Functional_Test.Button_PLC_Functional_Test_10 )
   END_RUNG
   RUNG wire#w1
      Contact( #In_Functional_Test.Electrical_Current_Test_Approved_PLC_Functional_Test_10 )
      Coil( #Out_Functional_Test.Electrical_Current_Test_Approved_PLC_Functional_Test_10 )
   END_RUNG
   RUNG wire#w1
      Contact( #In_Functional_Test.Visual_Test_Approved_PLC_Functional_Test_10 )
      Coil( #Out_Functional_Test.Visual_Test_Approved_PLC_Functional_Test_10 )
   END_RUNG
   RUNG wire#w1
      Move(in := #In_Functional_Test.Electrical_Current_Read_PLC_Functional_Test_10, out1 => #Out_Functional_Test.Electrical_Current_Read_PLC_Functional_Test_10)
   END_RUNG
   RUNG wire#w1
      Contact( #In_Functional_Test.Life_Trigger_PLC_Functional_Test_12 )
      Coil( #Out_Functional_Test.Life_Trigger_PLC_Functional_Test_12 )
   END_RUNG
   RUNG wire#w1
      Contact( #In_Functional_Test.Star_Test_PLC_Functional_Test_12 )
      Coil( #Out_Functional_Test.Star_Test_PLC_Functional_Test_12 )
   END_RUNG
   RUNG wire#w1
      Contact( #In_Functional_Test.Button_PLC_Functional_Test_12 )
      Coil( #Out_Functional_Test.Button_PLC_Functional_Test_12 )
   END_RUNG
   RUNG wire#w1
      Contact( #In_Functional_Test.Electrical_Current_Test_Approved_PLC_Functional_Test_12 )
      Coil( #Out_Functional_Test.Electrical_Current_Test_Approved_PLC_Functional_Test_12 )
   END_RUNG
   RUNG wire#w1
      Contact( #In_Functional_Test.Visual_Test_Approved_PLC_Functional_Test_12 )
      Coil( #Out_Functional_Test.Visual_Test_Approved_PLC_Functional_Test_12 )
   END_RUNG
   RUNG wire#w1
      Move(in := #In_Functional_Test.Electrical_Current_Read_PLC_Functional_Test_12, out1 => #Out_Functional_Test.Electrical_Current_Read_PLC_Functional_Test_12)
   END_RUNG
   RUNG wire#w1
      Contact( #In_Functional_Test.Life_Trigger_PLC_Functional_Test_14 )
      Coil( #Out_Functional_Test.Life_Trigger_PLC_Functional_Test_14 )
   END_RUNG
   RUNG wire#w1
      Contact( #In_Functional_Test.Star_Test_PLC_Functional_Test_14 )
      Coil( #Out_Functional_Test.Star_Test_PLC_Functional_Test_14 )
   END_RUNG
   RUNG wire#w1
      Contact( #In_Functional_Test.Button_PLC_Functional_Test_14 )
      Coil( #Out_Functional_Test.Button_PLC_Functional_Test_14 )
   END_RUNG
   RUNG wire#w1
      Contact( #In_Functional_Test.Electrical_Current_Test_Approved_PLC_Functional_Test_14 )
      Coil( #Out_Functional_Test.Electrical_Current_Test_Approved_PLC_Functional_Test_14 )
   END_RUNG
   RUNG wire#w1
      Contact( #In_Functional_Test.Visual_Test_Approved_PLC_Functional_Test_14 )
      Coil( #Out_Functional_Test.Visual_Test_Approved_PLC_Functional_Test_14 )
   END_RUNG
   RUNG wire#w1
      Move(in := #In_Functional_Test.Electrical_Current_Read_PLC_Functional_Test_14, out1 => #Out_Functional_Test.Electrical_Current_Read_PLC_Functional_Test_14)
   END_RUNG
   RUNG wire#w1
      Contact( #In_Functional_Test.Life_Trigger_PLC_Functional_Test_16 )
      Coil( #Out_Functional_Test.Life_Trigger_PLC_Functional_Test_16 )
   END_RUNG
   RUNG wire#w1
      Contact( #In_Functional_Test.Star_Test_PLC_Functional_Test_16 )
      Coil( #Out_Functional_Test.Star_Test_PLC_Functional_Test_16 )
   END_RUNG
   RUNG wire#w1
      Contact( #In_Functional_Test.Button_PLC_Functional_Test_16 )
      Coil( #Out_Functional_Test.Button_PLC_Functional_Test_16 )
   END_RUNG
   RUNG wire#w1
      Contact( #In_Functional_Test.Electrical_Current_Test_Approved_PLC_Functional_Test_16 )
      Coil( #Out_Functional_Test.Electrical_Current_Test_Approved_PLC_Functional_Test_16 )
   END_RUNG
   RUNG wire#w1
      Contact( #In_Functional_Test.Visual_Test_Approved_PLC_Functional_Test_16 )
      Coil( #Out_Functional_Test.Visual_Test_Approved_PLC_Functional_Test_16 )
   END_RUNG
   RUNG wire#w1
      Move(in := #In_Functional_Test.Electrical_Current_Read_PLC_Functional_Test_16, out1 => #Out_Functional_Test.Electrical_Current_Read_PLC_Functional_Test_16)
   END_RUNG
   RUNG wire#w1
      Contact( #In_Functional_Test.Life_Trigger_PLC_Functional_Test_18 )
      Coil( #Out_Functional_Test.Life_Trigger_PLC_Functional_Test_18 )
   END_RUNG
   RUNG wire#w1
      Contact( #In_Functional_Test.Star_Test_PLC_Functional_Test_18 )
      Coil( #Out_Functional_Test.Star_Test_PLC_Functional_Test_18 )
   END_RUNG
   RUNG wire#w1
      Contact( #In_Functional_Test.Button_PLC_Functional_Test_18 )
      Coil( #Out_Functional_Test.Button_PLC_Functional_Test_18 )
   END_RUNG
   RUNG wire#w1
      Contact( #In_Functional_Test.Electrical_Current_Test_Approved_PLC_Functional_Test_18 )
      Coil( #Out_Functional_Test.Electrical_Current_Test_Approved_PLC_Functional_Test_18 )
   END_RUNG
   RUNG wire#w1
      Contact( #In_Functional_Test.Visual_Test_Approved_PLC_Functional_Test_18 )
      Coil( #Out_Functional_Test.Visual_Test_Approved_PLC_Functional_Test_18 )
   END_RUNG
   RUNG wire#w1
      Move(in := #In_Functional_Test.Electrical_Current_Read_PLC_Functional_Test_18, out1 => #Out_Functional_Test.Electrical_Current_Read_PLC_Functional_Test_18)
   END_RUNG
   RUNG wire#w1
      Contact( #In_Functional_Test.Life_Trigger_PLC_Functional_Test_20 )
      Coil( #Out_Functional_Test.Life_Trigger_PLC_Functional_Test_20 )
   END_RUNG
   RUNG wire#w1
      Contact( #In_Functional_Test.Star_Test_PLC_Functional_Test_20 )
      Coil( #Out_Functional_Test.Star_Test_PLC_Functional_Test_20 )
   END_RUNG
   RUNG wire#w1
      Contact( #In_Functional_Test.Button_PLC_Functional_Test_20 )
      Coil( #Out_Functional_Test.Button_PLC_Functional_Test_20 )
   END_RUNG
   RUNG wire#w1
      Contact( #In_Functional_Test.Electrical_Current_Test_Approved_PLC_Functional_Test_20 )
      Coil( #Out_Functional_Test.Electrical_Current_Test_Approved_PLC_Functional_Test_20 )
   END_RUNG
   RUNG wire#w1
      Contact( #In_Functional_Test.Visual_Test_Approved_PLC_Functional_Test_20 )
      Coil( #Out_Functional_Test.Visual_Test_Approved_PLC_Functional_Test_20 )
   END_RUNG
   RUNG wire#w1
      Move(in := #In_Functional_Test.Electrical_Current_Read_PLC_Functional_Test_20, out1 => #Out_Functional_Test.Electrical_Current_Read_PLC_Functional_Test_20)
   END_RUNG
   RUNG wire#w1
      Contact( #In_Functional_Test.Life_Trigger_PLC_Functional_Test_22 )
      Coil( #Out_Functional_Test.Life_Trigger_PLC_Functional_Test_22 )
   END_RUNG
   RUNG wire#w1
      Contact( #In_Functional_Test.Star_Test_PLC_Functional_Test_22 )
      Coil( #Out_Functional_Test.Star_Test_PLC_Functional_Test_22 )
   END_RUNG
   RUNG wire#w1
      Contact( #In_Functional_Test.Button_PLC_Functional_Test_22 )
      Coil( #Out_Functional_Test.Button_PLC_Functional_Test_22 )
   END_RUNG
   RUNG wire#w1
      Contact( #In_Functional_Test.Electrical_Current_Test_Approved_PLC_Functional_Test_22 )
      Coil( #Out_Functional_Test.Electrical_Current_Test_Approved_PLC_Functional_Test_22 )
   END_RUNG
   RUNG wire#w1
      Contact( #In_Functional_Test.Visual_Test_Approved_PLC_Functional_Test_22 )
      Coil( #Out_Functional_Test.Visual_Test_Approved_PLC_Functional_Test_22 )
   END_RUNG
   RUNG wire#w1
      Move(in := #In_Functional_Test.Electrical_Current_Read_PLC_Functional_Test_22, out1 => #Out_Functional_Test.Electrical_Current_Read_PLC_Functional_Test_22)
   END_RUNG
   RUNG wire#w1
      Contact( #In_Functional_Test.Life_Trigger_PLC_Functional_Test_24 )
      Coil( #Out_Functional_Test.Life_Trigger_PLC_Functional_Test_24 )
   END_RUNG
   RUNG wire#w1
      Contact( #In_Functional_Test.Star_Test_PLC_Functional_Test_24 )
      Coil( #Out_Functional_Test.Star_Test_PLC_Functional_Test_24 )
   END_RUNG
   RUNG wire#w1
      Contact( #In_Functional_Test.Button_PLC_Functional_Test_24 )
      Coil( #Out_Functional_Test.Button_PLC_Functional_Test_24 )
   END_RUNG
   RUNG wire#w1
      Contact( #In_Functional_Test.Electrical_Current_Test_Approved_PLC_Functional_Test_24 )
      Coil( #Out_Functional_Test.Electrical_Current_Test_Approved_PLC_Functional_Test_24 )
   END_RUNG
   RUNG wire#w1
      Contact( #In_Functional_Test.Visual_Test_Approved_PLC_Functional_Test_24 )
      Coil( #Out_Functional_Test.Visual_Test_Approved_PLC_Functional_Test_24 )
   END_RUNG
   RUNG wire#w1
      Move(in := #In_Functional_Test.Electrical_Current_Read_PLC_Functional_Test_24, out1 => #Out_Functional_Test.Electrical_Current_Read_PLC_Functional_Test_24)
   END_RUNG
   RUNG wire#w1
      Contact( #In_Functional_Test.Life_Trigger_PLC_Functional_Test_26 )
      Coil( #Out_Functional_Test.Life_Trigger_PLC_Functional_Test_26 )
   END_RUNG
   RUNG wire#w1
      Contact( #In_Functional_Test.Star_Test_PLC_Functional_Test_26 )
      Coil( #Out_Functional_Test.Star_Test_PLC_Functional_Test_26 )
   END_RUNG
   RUNG wire#w1
      Contact( #In_Functional_Test.Button_PLC_Functional_Test_26 )
      Coil( #Out_Functional_Test.Button_PLC_Functional_Test_26 )
   END_RUNG
   RUNG wire#w1
      Contact( #In_Functional_Test.Electrical_Current_Test_Approved_PLC_Functional_Test_26 )
      Coil( #Out_Functional_Test.Electrical_Current_Test_Approved_PLC_Functional_Test_26 )
   END_RUNG
   RUNG wire#w1
      Contact( #In_Functional_Test.Visual_Test_Approved_PLC_Functional_Test_26 )
      Coil( #Out_Functional_Test.Visual_Test_Approved_PLC_Functional_Test_26 )
   END_RUNG
   RUNG wire#w1
      Move(in := #In_Functional_Test.Electrical_Current_Read_PLC_Functional_Test_26, out1 => #Out_Functional_Test.Electrical_Current_Read_PLC_Functional_Test_26)
   END_RUNG
   RUNG wire#w1
      Contact( #In_Functional_Test.Life_Trigger_PLC_Functional_Test_28 )
      Coil( #Out_Functional_Test.Life_Trigger_PLC_Functional_Test_28 )
   END_RUNG
   RUNG wire#w1
      Contact( #In_Functional_Test.Star_Test_PLC_Functional_Test_28 )
      Coil( #Out_Functional_Test.Star_Test_PLC_Functional_Test_28 )
   END_RUNG
   RUNG wire#w1
      Contact( #In_Functional_Test.Button_PLC_Functional_Test_28 )
      Coil( #Out_Functional_Test.Button_PLC_Functional_Test_28 )
   END_RUNG
   RUNG wire#w1
      Contact( #In_Functional_Test.Electrical_Current_Test_Approved_PLC_Functional_Test_28 )
      Coil( #Out_Functional_Test.Electrical_Current_Test_Approved_PLC_Functional_Test_28 )
   END_RUNG
   RUNG wire#w1
      Contact( #In_Functional_Test.Visual_Test_Approved_PLC_Functional_Test_28 )
      Coil( #Out_Functional_Test.Visual_Test_Approved_PLC_Functional_Test_28 )
   END_RUNG
   RUNG wire#w1
      Move(in := #In_Functional_Test.Electrical_Current_Read_PLC_Functional_Test_28, out1 => #Out_Functional_Test.Electrical_Current_Read_PLC_Functional_Test_28)
   END_RUNG
   RUNG wire#w1
      Contact( #In_Functional_Test.Life_Trigger_PLC_Functional_Test_30 )
      Coil( #Out_Functional_Test.Life_Trigger_PLC_Functional_Test_30 )
   END_RUNG
   RUNG wire#w1
      Contact( #In_Functional_Test.Star_Test_PLC_Functional_Test_30 )
      Coil( #Out_Functional_Test.Star_Test_PLC_Functional_Test_30 )
   END_RUNG
   RUNG wire#w1
      Contact( #In_Functional_Test.Button_PLC_Functional_Test_30 )
      Coil( #Out_Functional_Test.Button_PLC_Functional_Test_30 )
   END_RUNG
   RUNG wire#w1
      Contact( #In_Functional_Test.Electrical_Current_Test_Approved_PLC_Functional_Test_30 )
      Coil( #Out_Functional_Test.Electrical_Current_Test_Approved_PLC_Functional_Test_30 )
   END_RUNG
   RUNG wire#w1
      Contact( #In_Functional_Test.Visual_Test_Approved_PLC_Functional_Test_30 )
      Coil( #Out_Functional_Test.Visual_Test_Approved_PLC_Functional_Test_30 )
   END_RUNG
   RUNG wire#w1
      Move(in := #In_Functional_Test.Electrical_Current_Read_PLC_Functional_Test_30, out1 => #Out_Functional_Test.Electrical_Current_Read_PLC_Functional_Test_30)
   END_RUNG
   // the same network as SCL:
   #_w1 := #Test_Station = 8;
   #Out_Functional_Test.Life_Trigger_PLC_Functional_Test_8 := #_w1 AND #Life_Trigger;
   #Out_Functional_Test.Star_Test_PLC_Functional_Test_8 := #_w1 AND #Star_Test;
   #Out_Functional_Test.Button_PLC_Functional_Test_8 := #_w1 AND #Button_Start_Approve;
   #Out_Functional_Test.Electrical_Current_Test_Approved_PLC_Functional_Test_8 := #_w1 AND #Electrical_Current_Test_Approved;
   #Out_Functional_Test.Visual_Test_Approved_PLC_Functional_Test_8 := #_w1 AND #Visual_Test_Approved;
   #Reset_Functional_Test := #_w1 AND #In_Test_Parameters.Reset_PLC_Functional_Test_8;
   IF #_w1 THEN
       #Out_Functional_Test.Electrical_Current_Read_PLC_Functional_Test_8 := #Electrical_Current_Read;
   END_IF;
   #Out_Functional_Test.Life_Trigger_PLC_Functional_Test_10 := #_w1 AND #In_Functional_Test.Life_Trigger_PLC_Functional_Test_10;
   #Out_Functional_Test.Star_Test_PLC_Functional_Test_10 := #_w1 AND #In_Functional_Test.Star_Test_PLC_Functional_Test_10;
   #Out_Functional_Test.Button_PLC_Functional_Test_10 := #_w1 AND #In_Functional_Test.Button_PLC_Functional_Test_10;
   #Out_Functional_Test.Electrical_Current_Test_Approved_PLC_Functional_Test_10 := #_w1 AND #In_Functional_Test.Electrical_Current_Test_Approved_PLC_Functional_Test_10;
   #Out_Functional_Test.Visual_Test_Approved_PLC_Functional_Test_10 := #_w1 AND #In_Functional_Test.Visual_Test_Approved_PLC_Functional_Test_10;
   IF #_w1 THEN
       #Out_Functional_Test.Electrical_Current_Read_PLC_Functional_Test_10 := #In_Functional_Test.Electrical_Current_Read_PLC_Functional_Test_10;
   END_IF;
   #Out_Functional_Test.Life_Trigger_PLC_Functional_Test_12 := #_w1 AND #In_Functional_Test.Life_Trigger_PLC_Functional_Test_12;
   #Out_Functional_Test.Star_Test_PLC_Functional_Test_12 := #_w1 AND #In_Functional_Test.Star_Test_PLC_Functional_Test_12;
   #Out_Functional_Test.Button_PLC_Functional_Test_12 := #_w1 AND #In_Functional_Test.Button_PLC_Functional_Test_12;
   #Out_Functional_Test.Electrical_Current_Test_Approved_PLC_Functional_Test_12 := #_w1 AND #In_Functional_Test.Electrical_Current_Test_Approved_PLC_Functional_Test_12;
   #Out_Functional_Test.Visual_Test_Approved_PLC_Functional_Test_12 := #_w1 AND #In_Functional_Test.Visual_Test_Approved_PLC_Functional_Test_12;
   IF #_w1 THEN
       #Out_Functional_Test.Electrical_Current_Read_PLC_Functional_Test_12 := #In_Functional_Test.Electrical_Current_Read_PLC_Functional_Test_12;
   END_IF;
   #Out_Functional_Test.Life_Trigger_PLC_Functional_Test_14 := #_w1 AND #In_Functional_Test.Life_Trigger_PLC_Functional_Test_14;
   #Out_Functional_Test.Star_Test_PLC_Functional_Test_14 := #_w1 AND #In_Functional_Test.Star_Test_PLC_Functional_Test_14;
   #Out_Functional_Test.Button_PLC_Functional_Test_14 := #_w1 AND #In_Functional_Test.Button_PLC_Functional_Test_14;
   #Out_Functional_Test.Electrical_Current_Test_Approved_PLC_Functional_Test_14 := #_w1 AND #In_Functional_Test.Electrical_Current_Test_Approved_PLC_Functional_Test_14;
   #Out_Functional_Test.Visual_Test_Approved_PLC_Functional_Test_14 := #_w1 AND #In_Functional_Test.Visual_Test_Approved_PLC_Functional_Test_14;
   IF #_w1 THEN
       #Out_Functional_Test.Electrical_Current_Read_PLC_Functional_Test_14 := #In_Functional_Test.Electrical_Current_Read_PLC_Functional_Test_14;
   END_IF;
   #Out_Functional_Test.Life_Trigger_PLC_Functional_Test_16 := #_w1 AND #In_Functional_Test.Life_Trigger_PLC_Functional_Test_16;
   #Out_Functional_Test.Star_Test_PLC_Functional_Test_16 := #_w1 AND #In_Functional_Test.Star_Test_PLC_Functional_Test_16;
   #Out_Functional_Test.Button_PLC_Functional_Test_16 := #_w1 AND #In_Functional_Test.Button_PLC_Functional_Test_16;
   #Out_Functional_Test.Electrical_Current_Test_Approved_PLC_Functional_Test_16 := #_w1 AND #In_Functional_Test.Electrical_Current_Test_Approved_PLC_Functional_Test_16;
   #Out_Functional_Test.Visual_Test_Approved_PLC_Functional_Test_16 := #_w1 AND #In_Functional_Test.Visual_Test_Approved_PLC_Functional_Test_16;
   IF #_w1 THEN
       #Out_Functional_Test.Electrical_Current_Read_PLC_Functional_Test_16 := #In_Functional_Test.Electrical_Current_Read_PLC_Functional_Test_16;
   END_IF;
   #Out_Functional_Test.Life_Trigger_PLC_Functional_Test_18 := #_w1 AND #In_Functional_Test.Life_Trigger_PLC_Functional_Test_18;
   #Out_Functional_Test.Star_Test_PLC_Functional_Test_18 := #_w1 AND #In_Functional_Test.Star_Test_PLC_Functional_Test_18;
   #Out_Functional_Test.Button_PLC_Functional_Test_18 := #_w1 AND #In_Functional_Test.Button_PLC_Functional_Test_18;
   #Out_Functional_Test.Electrical_Current_Test_Approved_PLC_Functional_Test_18 := #_w1 AND #In_Functional_Test.Electrical_Current_Test_Approved_PLC_Functional_Test_18;
   #Out_Functional_Test.Visual_Test_Approved_PLC_Functional_Test_18 := #_w1 AND #In_Functional_Test.Visual_Test_Approved_PLC_Functional_Test_18;
   IF #_w1 THEN
       #Out_Functional_Test.Electrical_Current_Read_PLC_Functional_Test_18 := #In_Functional_Test.Electrical_Current_Read_PLC_Functional_Test_18;
   END_IF;
   #Out_Functional_Test.Life_Trigger_PLC_Functional_Test_20 := #_w1 AND #In_Functional_Test.Life_Trigger_PLC_Functional_Test_20;
   #Out_Functional_Test.Star_Test_PLC_Functional_Test_20 := #_w1 AND #In_Functional_Test.Star_Test_PLC_Functional_Test_20;
   #Out_Functional_Test.Button_PLC_Functional_Test_20 := #_w1 AND #In_Functional_Test.Button_PLC_Functional_Test_20;
   #Out_Functional_Test.Electrical_Current_Test_Approved_PLC_Functional_Test_20 := #_w1 AND #In_Functional_Test.Electrical_Current_Test_Approved_PLC_Functional_Test_20;
   #Out_Functional_Test.Visual_Test_Approved_PLC_Functional_Test_20 := #_w1 AND #In_Functional_Test.Visual_Test_Approved_PLC_Functional_Test_20;
   IF #_w1 THEN
       #Out_Functional_Test.Electrical_Current_Read_PLC_Functional_Test_20 := #In_Functional_Test.Electrical_Current_Read_PLC_Functional_Test_20;
   END_IF;
   #Out_Functional_Test.Life_Trigger_PLC_Functional_Test_22 := #_w1 AND #In_Functional_Test.Life_Trigger_PLC_Functional_Test_22;
   #Out_Functional_Test.Star_Test_PLC_Functional_Test_22 := #_w1 AND #In_Functional_Test.Star_Test_PLC_Functional_Test_22;
   #Out_Functional_Test.Button_PLC_Functional_Test_22 := #_w1 AND #In_Functional_Test.Button_PLC_Functional_Test_22;
   #Out_Functional_Test.Electrical_Current_Test_Approved_PLC_Functional_Test_22 := #_w1 AND #In_Functional_Test.Electrical_Current_Test_Approved_PLC_Functional_Test_22;
   #Out_Functional_Test.Visual_Test_Approved_PLC_Functional_Test_22 := #_w1 AND #In_Functional_Test.Visual_Test_Approved_PLC_Functional_Test_22;
   IF #_w1 THEN
       #Out_Functional_Test.Electrical_Current_Read_PLC_Functional_Test_22 := #In_Functional_Test.Electrical_Current_Read_PLC_Functional_Test_22;
   END_IF;
   #Out_Functional_Test.Life_Trigger_PLC_Functional_Test_24 := #_w1 AND #In_Functional_Test.Life_Trigger_PLC_Functional_Test_24;
   #Out_Functional_Test.Star_Test_PLC_Functional_Test_24 := #_w1 AND #In_Functional_Test.Star_Test_PLC_Functional_Test_24;
   #Out_Functional_Test.Button_PLC_Functional_Test_24 := #_w1 AND #In_Functional_Test.Button_PLC_Functional_Test_24;
   #Out_Functional_Test.Electrical_Current_Test_Approved_PLC_Functional_Test_24 := #_w1 AND #In_Functional_Test.Electrical_Current_Test_Approved_PLC_Functional_Test_24;
   #Out_Functional_Test.Visual_Test_Approved_PLC_Functional_Test_24 := #_w1 AND #In_Functional_Test.Visual_Test_Approved_PLC_Functional_Test_24;
   IF #_w1 THEN
       #Out_Functional_Test.Electrical_Current_Read_PLC_Functional_Test_24 := #In_Functional_Test.Electrical_Current_Read_PLC_Functional_Test_24;
   END_IF;
   #Out_Functional_Test.Life_Trigger_PLC_Functional_Test_26 := #_w1 AND #In_Functional_Test.Life_Trigger_PLC_Functional_Test_26;
   #Out_Functional_Test.Star_Test_PLC_Functional_Test_26 := #_w1 AND #In_Functional_Test.Star_Test_PLC_Functional_Test_26;
   #Out_Functional_Test.Button_PLC_Functional_Test_26 := #_w1 AND #In_Functional_Test.Button_PLC_Functional_Test_26;
   #Out_Functional_Test.Electrical_Current_Test_Approved_PLC_Functional_Test_26 := #_w1 AND #In_Functional_Test.Electrical_Current_Test_Approved_PLC_Functional_Test_26;
   #Out_Functional_Test.Visual_Test_Approved_PLC_Functional_Test_26 := #_w1 AND #In_Functional_Test.Visual_Test_Approved_PLC_Functional_Test_26;
   IF #_w1 THEN
       #Out_Functional_Test.Electrical_Current_Read_PLC_Functional_Test_26 := #In_Functional_Test.Electrical_Current_Read_PLC_Functional_Test_26;
   END_IF;
   #Out_Functional_Test.Life_Trigger_PLC_Functional_Test_28 := #_w1 AND #In_Functional_Test.Life_Trigger_PLC_Functional_Test_28;
   #Out_Functional_Test.Star_Test_PLC_Functional_Test_28 := #_w1 AND #In_Functional_Test.Star_Test_PLC_Functional_Test_28;
   #Out_Functional_Test.Button_PLC_Functional_Test_28 := #_w1 AND #In_Functional_Test.Button_PLC_Functional_Test_28;
   #Out_Functional_Test.Electrical_Current_Test_Approved_PLC_Functional_Test_28 := #_w1 AND #In_Functional_Test.Electrical_Current_Test_Approved_PLC_Functional_Test_28;
   #Out_Functional_Test.Visual_Test_Approved_PLC_Functional_Test_28 := #_w1 AND #In_Functional_Test.Visual_Test_Approved_PLC_Functional_Test_28;
   IF #_w1 THEN
       #Out_Functional_Test.Electrical_Current_Read_PLC_Functional_Test_28 := #In_Functional_Test.Electrical_Current_Read_PLC_Functional_Test_28;
   END_IF;
   #Out_Functional_Test.Life_Trigger_PLC_Functional_Test_30 := #_w1 AND #In_Functional_Test.Life_Trigger_PLC_Functional_Test_30;
   #Out_Functional_Test.Star_Test_PLC_Functional_Test_30 := #_w1 AND #In_Functional_Test.Star_Test_PLC_Functional_Test_30;
   #Out_Functional_Test.Button_PLC_Functional_Test_30 := #_w1 AND #In_Functional_Test.Button_PLC_Functional_Test_30;
   #Out_Functional_Test.Electrical_Current_Test_Approved_PLC_Functional_Test_30 := #_w1 AND #In_Functional_Test.Electrical_Current_Test_Approved_PLC_Functional_Test_30;
   #Out_Functional_Test.Visual_Test_Approved_PLC_Functional_Test_30 := #_w1 AND #In_Functional_Test.Visual_Test_Approved_PLC_Functional_Test_30;
   IF #_w1 THEN
       #Out_Functional_Test.Electrical_Current_Read_PLC_Functional_Test_30 := #In_Functional_Test.Electrical_Current_Read_PLC_Functional_Test_30;
   END_IF;
END_REGION

REGION Network 6: Functional Test Station 10
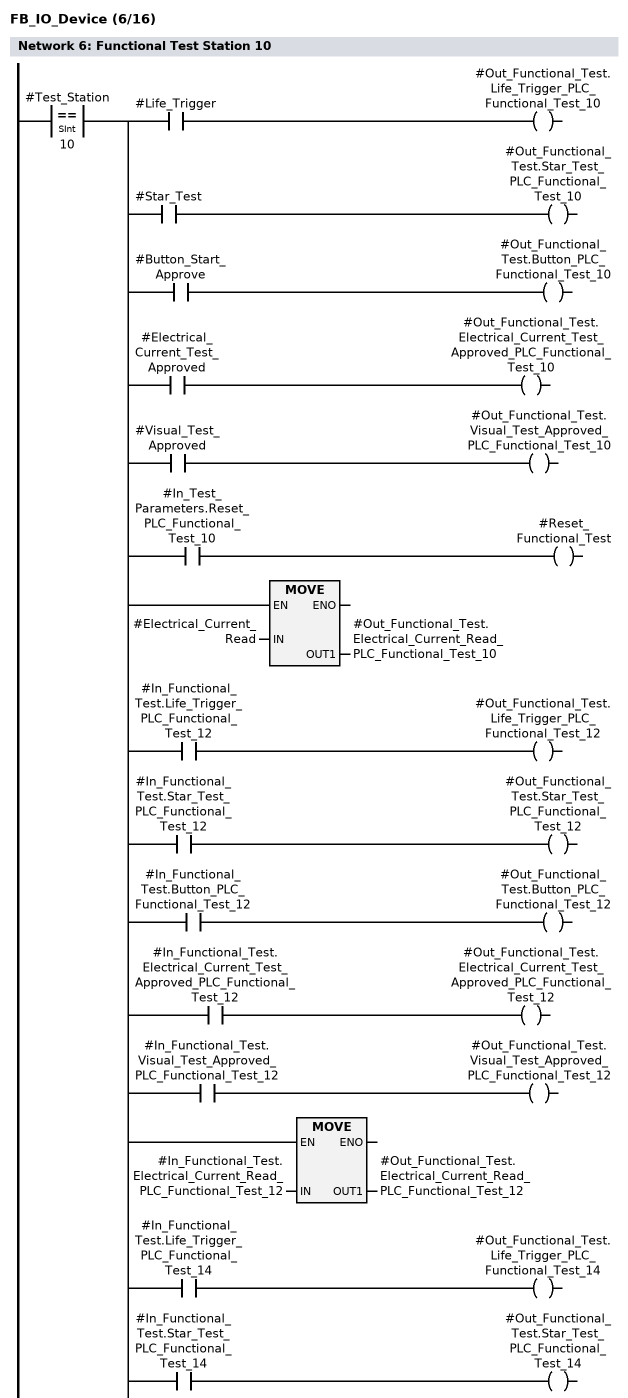
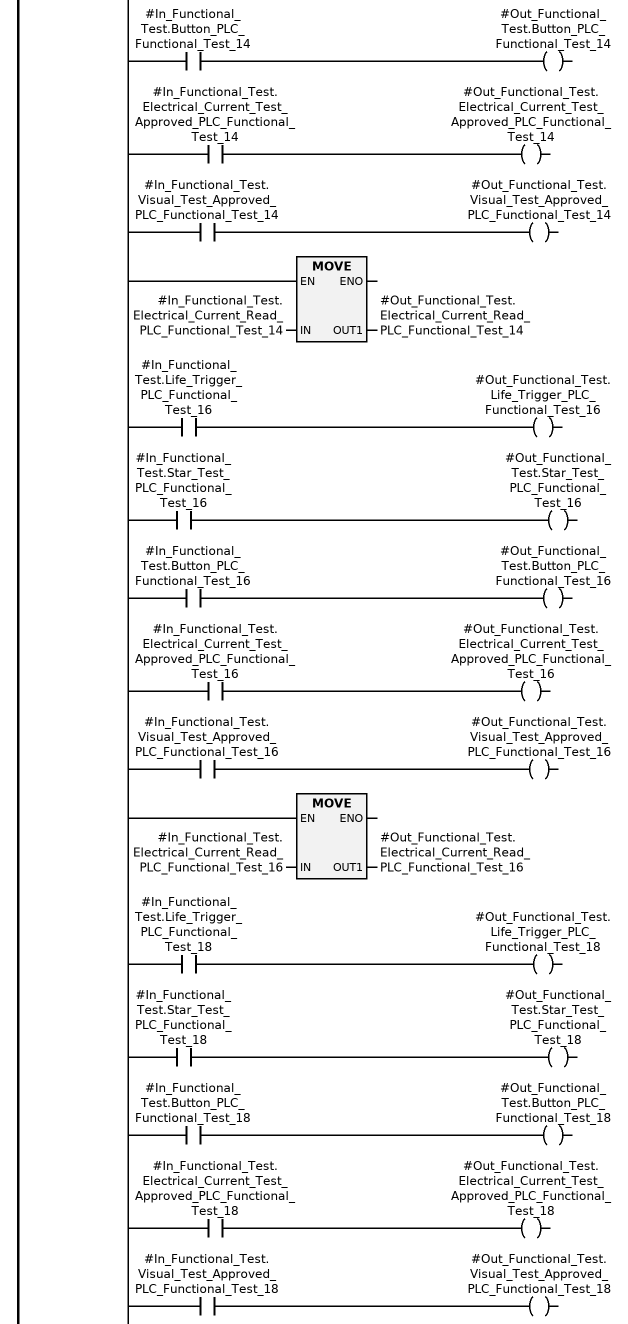
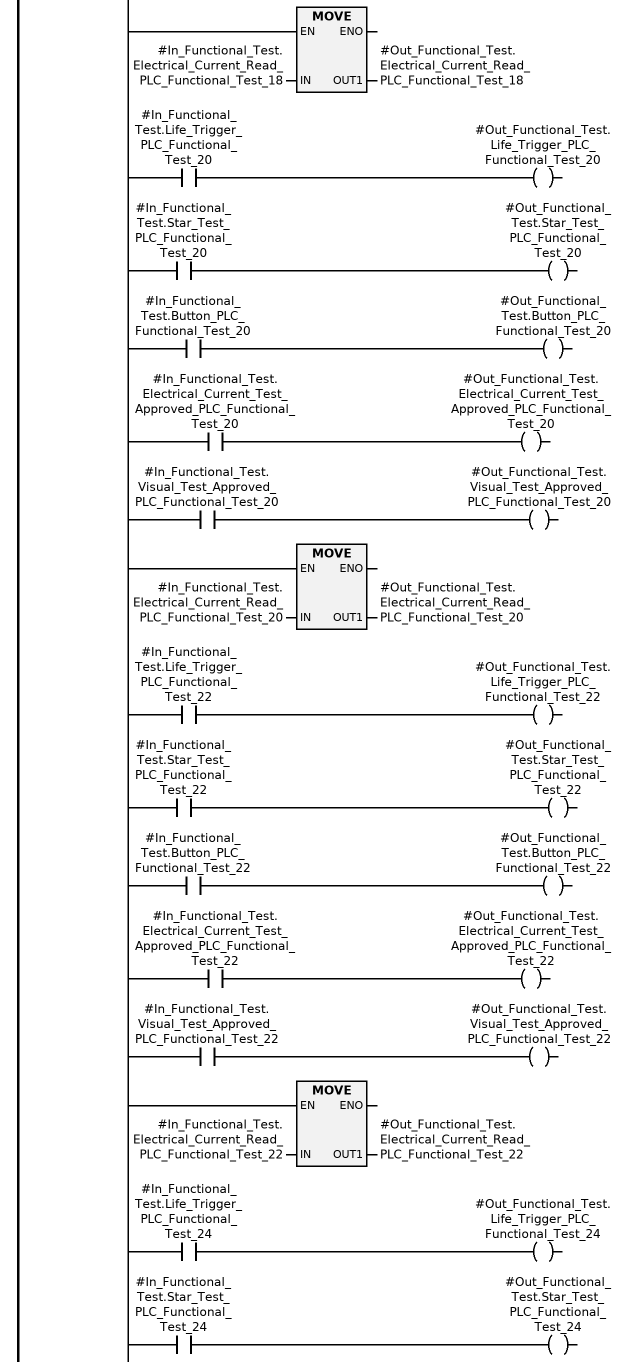
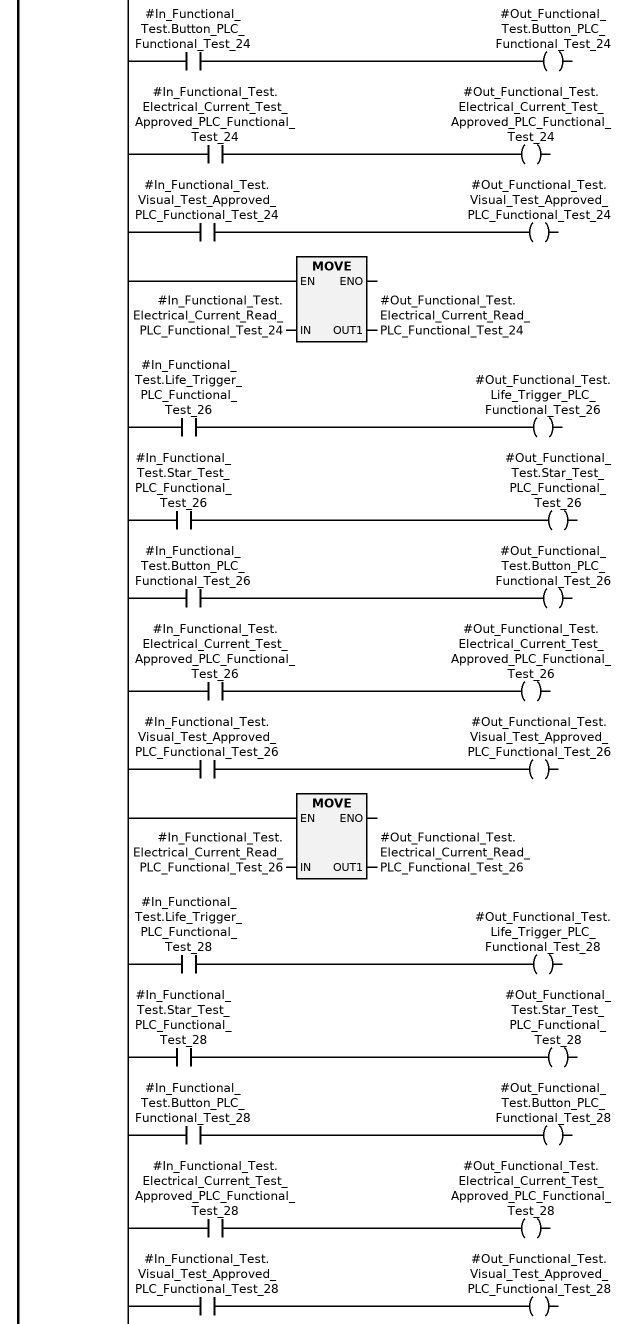
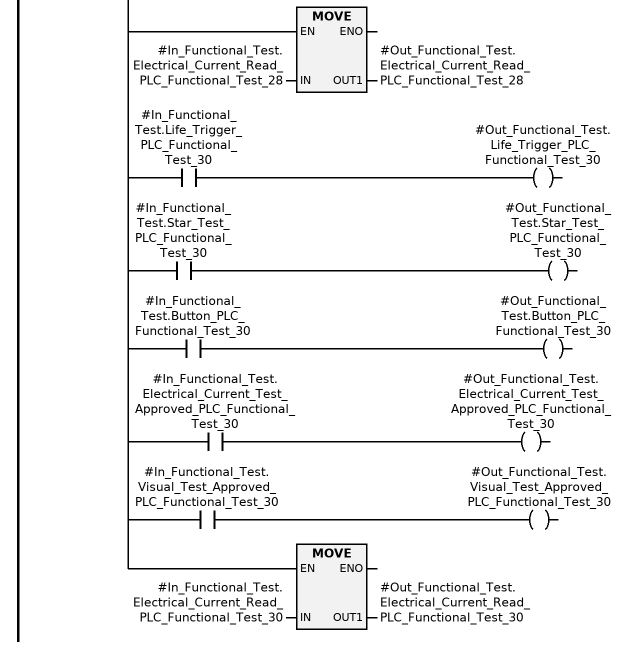
   RUNG wire#powerrail
      { S7_Templates := "SrcType := SInt" } EQ_Contact(in1 := #Test_Station, in2 := 10)
      wire#w1
      Contact( #Life_Trigger )
      Coil( #Out_Functional_Test.Life_Trigger_PLC_Functional_Test_10 )
   END_RUNG
   RUNG wire#w1
      Contact( #Star_Test )
      Coil( #Out_Functional_Test.Star_Test_PLC_Functional_Test_10 )
   END_RUNG
   RUNG wire#w1
      Contact( #Button_Start_Approve )
      Coil( #Out_Functional_Test.Button_PLC_Functional_Test_10 )
   END_RUNG
   RUNG wire#w1
      Contact( #Electrical_Current_Test_Approved )
      Coil( #Out_Functional_Test.Electrical_Current_Test_Approved_PLC_Functional_Test_10 )
   END_RUNG
   RUNG wire#w1
      Contact( #Visual_Test_Approved )
      Coil( #Out_Functional_Test.Visual_Test_Approved_PLC_Functional_Test_10 )
   END_RUNG
   RUNG wire#w1
      Contact( #In_Test_Parameters.Reset_PLC_Functional_Test_10 )
      Coil( #Reset_Functional_Test )
   END_RUNG
   RUNG wire#w1
      Move(in := #Electrical_Current_Read, out1 => #Out_Functional_Test.Electrical_Current_Read_PLC_Functional_Test_10)
   END_RUNG
   RUNG wire#w1
      Contact( #In_Functional_Test.Life_Trigger_PLC_Functional_Test_12 )
      Coil( #Out_Functional_Test.Life_Trigger_PLC_Functional_Test_12 )
   END_RUNG
   RUNG wire#w1
      Contact( #In_Functional_Test.Star_Test_PLC_Functional_Test_12 )
      Coil( #Out_Functional_Test.Star_Test_PLC_Functional_Test_12 )
   END_RUNG
   RUNG wire#w1
      Contact( #In_Functional_Test.Button_PLC_Functional_Test_12 )
      Coil( #Out_Functional_Test.Button_PLC_Functional_Test_12 )
   END_RUNG
   RUNG wire#w1
      Contact( #In_Functional_Test.Electrical_Current_Test_Approved_PLC_Functional_Test_12 )
      Coil( #Out_Functional_Test.Electrical_Current_Test_Approved_PLC_Functional_Test_12 )
   END_RUNG
   RUNG wire#w1
      Contact( #In_Functional_Test.Visual_Test_Approved_PLC_Functional_Test_12 )
      Coil( #Out_Functional_Test.Visual_Test_Approved_PLC_Functional_Test_12 )
   END_RUNG
   RUNG wire#w1
      Move(in := #In_Functional_Test.Electrical_Current_Read_PLC_Functional_Test_12, out1 => #Out_Functional_Test.Electrical_Current_Read_PLC_Functional_Test_12)
   END_RUNG
   RUNG wire#w1
      Contact( #In_Functional_Test.Life_Trigger_PLC_Functional_Test_14 )
      Coil( #Out_Functional_Test.Life_Trigger_PLC_Functional_Test_14 )
   END_RUNG
   RUNG wire#w1
      Contact( #In_Functional_Test.Star_Test_PLC_Functional_Test_14 )
      Coil( #Out_Functional_Test.Star_Test_PLC_Functional_Test_14 )
   END_RUNG
   RUNG wire#w1
      Contact( #In_Functional_Test.Button_PLC_Functional_Test_14 )
      Coil( #Out_Functional_Test.Button_PLC_Functional_Test_14 )
   END_RUNG
   RUNG wire#w1
      Contact( #In_Functional_Test.Electrical_Current_Test_Approved_PLC_Functional_Test_14 )
      Coil( #Out_Functional_Test.Electrical_Current_Test_Approved_PLC_Functional_Test_14 )
   END_RUNG
   RUNG wire#w1
      Contact( #In_Functional_Test.Visual_Test_Approved_PLC_Functional_Test_14 )
      Coil( #Out_Functional_Test.Visual_Test_Approved_PLC_Functional_Test_14 )
   END_RUNG
   RUNG wire#w1
      Move(in := #In_Functional_Test.Electrical_Current_Read_PLC_Functional_Test_14, out1 => #Out_Functional_Test.Electrical_Current_Read_PLC_Functional_Test_14)
   END_RUNG
   RUNG wire#w1
      Contact( #In_Functional_Test.Life_Trigger_PLC_Functional_Test_16 )
      Coil( #Out_Functional_Test.Life_Trigger_PLC_Functional_Test_16 )
   END_RUNG
   RUNG wire#w1
      Contact( #In_Functional_Test.Star_Test_PLC_Functional_Test_16 )
      Coil( #Out_Functional_Test.Star_Test_PLC_Functional_Test_16 )
   END_RUNG
   RUNG wire#w1
      Contact( #In_Functional_Test.Button_PLC_Functional_Test_16 )
      Coil( #Out_Functional_Test.Button_PLC_Functional_Test_16 )
   END_RUNG
   RUNG wire#w1
      Contact( #In_Functional_Test.Electrical_Current_Test_Approved_PLC_Functional_Test_16 )
      Coil( #Out_Functional_Test.Electrical_Current_Test_Approved_PLC_Functional_Test_16 )
   END_RUNG
   RUNG wire#w1
      Contact( #In_Functional_Test.Visual_Test_Approved_PLC_Functional_Test_16 )
      Coil( #Out_Functional_Test.Visual_Test_Approved_PLC_Functional_Test_16 )
   END_RUNG
   RUNG wire#w1
      Move(in := #In_Functional_Test.Electrical_Current_Read_PLC_Functional_Test_16, out1 => #Out_Functional_Test.Electrical_Current_Read_PLC_Functional_Test_16)
   END_RUNG
   RUNG wire#w1
      Contact( #In_Functional_Test.Life_Trigger_PLC_Functional_Test_18 )
      Coil( #Out_Functional_Test.Life_Trigger_PLC_Functional_Test_18 )
   END_RUNG
   RUNG wire#w1
      Contact( #In_Functional_Test.Star_Test_PLC_Functional_Test_18 )
      Coil( #Out_Functional_Test.Star_Test_PLC_Functional_Test_18 )
   END_RUNG
   RUNG wire#w1
      Contact( #In_Functional_Test.Button_PLC_Functional_Test_18 )
      Coil( #Out_Functional_Test.Button_PLC_Functional_Test_18 )
   END_RUNG
   RUNG wire#w1
      Contact( #In_Functional_Test.Electrical_Current_Test_Approved_PLC_Functional_Test_18 )
      Coil( #Out_Functional_Test.Electrical_Current_Test_Approved_PLC_Functional_Test_18 )
   END_RUNG
   RUNG wire#w1
      Contact( #In_Functional_Test.Visual_Test_Approved_PLC_Functional_Test_18 )
      Coil( #Out_Functional_Test.Visual_Test_Approved_PLC_Functional_Test_18 )
   END_RUNG
   RUNG wire#w1
      Move(in := #In_Functional_Test.Electrical_Current_Read_PLC_Functional_Test_18, out1 => #Out_Functional_Test.Electrical_Current_Read_PLC_Functional_Test_18)
   END_RUNG
   RUNG wire#w1
      Contact( #In_Functional_Test.Life_Trigger_PLC_Functional_Test_20 )
      Coil( #Out_Functional_Test.Life_Trigger_PLC_Functional_Test_20 )
   END_RUNG
   RUNG wire#w1
      Contact( #In_Functional_Test.Star_Test_PLC_Functional_Test_20 )
      Coil( #Out_Functional_Test.Star_Test_PLC_Functional_Test_20 )
   END_RUNG
   RUNG wire#w1
      Contact( #In_Functional_Test.Button_PLC_Functional_Test_20 )
      Coil( #Out_Functional_Test.Button_PLC_Functional_Test_20 )
   END_RUNG
   RUNG wire#w1
      Contact( #In_Functional_Test.Electrical_Current_Test_Approved_PLC_Functional_Test_20 )
      Coil( #Out_Functional_Test.Electrical_Current_Test_Approved_PLC_Functional_Test_20 )
   END_RUNG
   RUNG wire#w1
      Contact( #In_Functional_Test.Visual_Test_Approved_PLC_Functional_Test_20 )
      Coil( #Out_Functional_Test.Visual_Test_Approved_PLC_Functional_Test_20 )
   END_RUNG
   RUNG wire#w1
      Move(in := #In_Functional_Test.Electrical_Current_Read_PLC_Functional_Test_20, out1 => #Out_Functional_Test.Electrical_Current_Read_PLC_Functional_Test_20)
   END_RUNG
   RUNG wire#w1
      Contact( #In_Functional_Test.Life_Trigger_PLC_Functional_Test_22 )
      Coil( #Out_Functional_Test.Life_Trigger_PLC_Functional_Test_22 )
   END_RUNG
   RUNG wire#w1
      Contact( #In_Functional_Test.Star_Test_PLC_Functional_Test_22 )
      Coil( #Out_Functional_Test.Star_Test_PLC_Functional_Test_22 )
   END_RUNG
   RUNG wire#w1
      Contact( #In_Functional_Test.Button_PLC_Functional_Test_22 )
      Coil( #Out_Functional_Test.Button_PLC_Functional_Test_22 )
   END_RUNG
   RUNG wire#w1
      Contact( #In_Functional_Test.Electrical_Current_Test_Approved_PLC_Functional_Test_22 )
      Coil( #Out_Functional_Test.Electrical_Current_Test_Approved_PLC_Functional_Test_22 )
   END_RUNG
   RUNG wire#w1
      Contact( #In_Functional_Test.Visual_Test_Approved_PLC_Functional_Test_22 )
      Coil( #Out_Functional_Test.Visual_Test_Approved_PLC_Functional_Test_22 )
   END_RUNG
   RUNG wire#w1
      Move(in := #In_Functional_Test.Electrical_Current_Read_PLC_Functional_Test_22, out1 => #Out_Functional_Test.Electrical_Current_Read_PLC_Functional_Test_22)
   END_RUNG
   RUNG wire#w1
      Contact( #In_Functional_Test.Life_Trigger_PLC_Functional_Test_24 )
      Coil( #Out_Functional_Test.Life_Trigger_PLC_Functional_Test_24 )
   END_RUNG
   RUNG wire#w1
      Contact( #In_Functional_Test.Star_Test_PLC_Functional_Test_24 )
      Coil( #Out_Functional_Test.Star_Test_PLC_Functional_Test_24 )
   END_RUNG
   RUNG wire#w1
      Contact( #In_Functional_Test.Button_PLC_Functional_Test_24 )
      Coil( #Out_Functional_Test.Button_PLC_Functional_Test_24 )
   END_RUNG
   RUNG wire#w1
      Contact( #In_Functional_Test.Electrical_Current_Test_Approved_PLC_Functional_Test_24 )
      Coil( #Out_Functional_Test.Electrical_Current_Test_Approved_PLC_Functional_Test_24 )
   END_RUNG
   RUNG wire#w1
      Contact( #In_Functional_Test.Visual_Test_Approved_PLC_Functional_Test_24 )
      Coil( #Out_Functional_Test.Visual_Test_Approved_PLC_Functional_Test_24 )
   END_RUNG
   RUNG wire#w1
      Move(in := #In_Functional_Test.Electrical_Current_Read_PLC_Functional_Test_24, out1 => #Out_Functional_Test.Electrical_Current_Read_PLC_Functional_Test_24)
   END_RUNG
   RUNG wire#w1
      Contact( #In_Functional_Test.Life_Trigger_PLC_Functional_Test_26 )
      Coil( #Out_Functional_Test.Life_Trigger_PLC_Functional_Test_26 )
   END_RUNG
   RUNG wire#w1
      Contact( #In_Functional_Test.Star_Test_PLC_Functional_Test_26 )
      Coil( #Out_Functional_Test.Star_Test_PLC_Functional_Test_26 )
   END_RUNG
   RUNG wire#w1
      Contact( #In_Functional_Test.Button_PLC_Functional_Test_26 )
      Coil( #Out_Functional_Test.Button_PLC_Functional_Test_26 )
   END_RUNG
   RUNG wire#w1
      Contact( #In_Functional_Test.Electrical_Current_Test_Approved_PLC_Functional_Test_26 )
      Coil( #Out_Functional_Test.Electrical_Current_Test_Approved_PLC_Functional_Test_26 )
   END_RUNG
   RUNG wire#w1
      Contact( #In_Functional_Test.Visual_Test_Approved_PLC_Functional_Test_26 )
      Coil( #Out_Functional_Test.Visual_Test_Approved_PLC_Functional_Test_26 )
   END_RUNG
   RUNG wire#w1
      Move(in := #In_Functional_Test.Electrical_Current_Read_PLC_Functional_Test_26, out1 => #Out_Functional_Test.Electrical_Current_Read_PLC_Functional_Test_26)
   END_RUNG
   RUNG wire#w1
      Contact( #In_Functional_Test.Life_Trigger_PLC_Functional_Test_28 )
      Coil( #Out_Functional_Test.Life_Trigger_PLC_Functional_Test_28 )
   END_RUNG
   RUNG wire#w1
      Contact( #In_Functional_Test.Star_Test_PLC_Functional_Test_28 )
      Coil( #Out_Functional_Test.Star_Test_PLC_Functional_Test_28 )
   END_RUNG
   RUNG wire#w1
      Contact( #In_Functional_Test.Button_PLC_Functional_Test_28 )
      Coil( #Out_Functional_Test.Button_PLC_Functional_Test_28 )
   END_RUNG
   RUNG wire#w1
      Contact( #In_Functional_Test.Electrical_Current_Test_Approved_PLC_Functional_Test_28 )
      Coil( #Out_Functional_Test.Electrical_Current_Test_Approved_PLC_Functional_Test_28 )
   END_RUNG
   RUNG wire#w1
      Contact( #In_Functional_Test.Visual_Test_Approved_PLC_Functional_Test_28 )
      Coil( #Out_Functional_Test.Visual_Test_Approved_PLC_Functional_Test_28 )
   END_RUNG
   RUNG wire#w1
      Move(in := #In_Functional_Test.Electrical_Current_Read_PLC_Functional_Test_28, out1 => #Out_Functional_Test.Electrical_Current_Read_PLC_Functional_Test_28)
   END_RUNG
   RUNG wire#w1
      Contact( #In_Functional_Test.Life_Trigger_PLC_Functional_Test_30 )
      Coil( #Out_Functional_Test.Life_Trigger_PLC_Functional_Test_30 )
   END_RUNG
   RUNG wire#w1
      Contact( #In_Functional_Test.Star_Test_PLC_Functional_Test_30 )
      Coil( #Out_Functional_Test.Star_Test_PLC_Functional_Test_30 )
   END_RUNG
   RUNG wire#w1
      Contact( #In_Functional_Test.Button_PLC_Functional_Test_30 )
      Coil( #Out_Functional_Test.Button_PLC_Functional_Test_30 )
   END_RUNG
   RUNG wire#w1
      Contact( #In_Functional_Test.Electrical_Current_Test_Approved_PLC_Functional_Test_30 )
      Coil( #Out_Functional_Test.Electrical_Current_Test_Approved_PLC_Functional_Test_30 )
   END_RUNG
   RUNG wire#w1
      Contact( #In_Functional_Test.Visual_Test_Approved_PLC_Functional_Test_30 )
      Coil( #Out_Functional_Test.Visual_Test_Approved_PLC_Functional_Test_30 )
   END_RUNG
   RUNG wire#w1
      Move(in := #In_Functional_Test.Electrical_Current_Read_PLC_Functional_Test_30, out1 => #Out_Functional_Test.Electrical_Current_Read_PLC_Functional_Test_30)
   END_RUNG
   // the same network as SCL:
   #_w1 := #Test_Station = 10;
   #Out_Functional_Test.Life_Trigger_PLC_Functional_Test_10 := #_w1 AND #Life_Trigger;
   #Out_Functional_Test.Star_Test_PLC_Functional_Test_10 := #_w1 AND #Star_Test;
   #Out_Functional_Test.Button_PLC_Functional_Test_10 := #_w1 AND #Button_Start_Approve;
   #Out_Functional_Test.Electrical_Current_Test_Approved_PLC_Functional_Test_10 := #_w1 AND #Electrical_Current_Test_Approved;
   #Out_Functional_Test.Visual_Test_Approved_PLC_Functional_Test_10 := #_w1 AND #Visual_Test_Approved;
   #Reset_Functional_Test := #_w1 AND #In_Test_Parameters.Reset_PLC_Functional_Test_10;
   IF #_w1 THEN
       #Out_Functional_Test.Electrical_Current_Read_PLC_Functional_Test_10 := #Electrical_Current_Read;
   END_IF;
   #Out_Functional_Test.Life_Trigger_PLC_Functional_Test_12 := #_w1 AND #In_Functional_Test.Life_Trigger_PLC_Functional_Test_12;
   #Out_Functional_Test.Star_Test_PLC_Functional_Test_12 := #_w1 AND #In_Functional_Test.Star_Test_PLC_Functional_Test_12;
   #Out_Functional_Test.Button_PLC_Functional_Test_12 := #_w1 AND #In_Functional_Test.Button_PLC_Functional_Test_12;
   #Out_Functional_Test.Electrical_Current_Test_Approved_PLC_Functional_Test_12 := #_w1 AND #In_Functional_Test.Electrical_Current_Test_Approved_PLC_Functional_Test_12;
   #Out_Functional_Test.Visual_Test_Approved_PLC_Functional_Test_12 := #_w1 AND #In_Functional_Test.Visual_Test_Approved_PLC_Functional_Test_12;
   IF #_w1 THEN
       #Out_Functional_Test.Electrical_Current_Read_PLC_Functional_Test_12 := #In_Functional_Test.Electrical_Current_Read_PLC_Functional_Test_12;
   END_IF;
   #Out_Functional_Test.Life_Trigger_PLC_Functional_Test_14 := #_w1 AND #In_Functional_Test.Life_Trigger_PLC_Functional_Test_14;
   #Out_Functional_Test.Star_Test_PLC_Functional_Test_14 := #_w1 AND #In_Functional_Test.Star_Test_PLC_Functional_Test_14;
   #Out_Functional_Test.Button_PLC_Functional_Test_14 := #_w1 AND #In_Functional_Test.Button_PLC_Functional_Test_14;
   #Out_Functional_Test.Electrical_Current_Test_Approved_PLC_Functional_Test_14 := #_w1 AND #In_Functional_Test.Electrical_Current_Test_Approved_PLC_Functional_Test_14;
   #Out_Functional_Test.Visual_Test_Approved_PLC_Functional_Test_14 := #_w1 AND #In_Functional_Test.Visual_Test_Approved_PLC_Functional_Test_14;
   IF #_w1 THEN
       #Out_Functional_Test.Electrical_Current_Read_PLC_Functional_Test_14 := #In_Functional_Test.Electrical_Current_Read_PLC_Functional_Test_14;
   END_IF;
   #Out_Functional_Test.Life_Trigger_PLC_Functional_Test_16 := #_w1 AND #In_Functional_Test.Life_Trigger_PLC_Functional_Test_16;
   #Out_Functional_Test.Star_Test_PLC_Functional_Test_16 := #_w1 AND #In_Functional_Test.Star_Test_PLC_Functional_Test_16;
   #Out_Functional_Test.Button_PLC_Functional_Test_16 := #_w1 AND #In_Functional_Test.Button_PLC_Functional_Test_16;
   #Out_Functional_Test.Electrical_Current_Test_Approved_PLC_Functional_Test_16 := #_w1 AND #In_Functional_Test.Electrical_Current_Test_Approved_PLC_Functional_Test_16;
   #Out_Functional_Test.Visual_Test_Approved_PLC_Functional_Test_16 := #_w1 AND #In_Functional_Test.Visual_Test_Approved_PLC_Functional_Test_16;
   IF #_w1 THEN
       #Out_Functional_Test.Electrical_Current_Read_PLC_Functional_Test_16 := #In_Functional_Test.Electrical_Current_Read_PLC_Functional_Test_16;
   END_IF;
   #Out_Functional_Test.Life_Trigger_PLC_Functional_Test_18 := #_w1 AND #In_Functional_Test.Life_Trigger_PLC_Functional_Test_18;
   #Out_Functional_Test.Star_Test_PLC_Functional_Test_18 := #_w1 AND #In_Functional_Test.Star_Test_PLC_Functional_Test_18;
   #Out_Functional_Test.Button_PLC_Functional_Test_18 := #_w1 AND #In_Functional_Test.Button_PLC_Functional_Test_18;
   #Out_Functional_Test.Electrical_Current_Test_Approved_PLC_Functional_Test_18 := #_w1 AND #In_Functional_Test.Electrical_Current_Test_Approved_PLC_Functional_Test_18;
   #Out_Functional_Test.Visual_Test_Approved_PLC_Functional_Test_18 := #_w1 AND #In_Functional_Test.Visual_Test_Approved_PLC_Functional_Test_18;
   IF #_w1 THEN
       #Out_Functional_Test.Electrical_Current_Read_PLC_Functional_Test_18 := #In_Functional_Test.Electrical_Current_Read_PLC_Functional_Test_18;
   END_IF;
   #Out_Functional_Test.Life_Trigger_PLC_Functional_Test_20 := #_w1 AND #In_Functional_Test.Life_Trigger_PLC_Functional_Test_20;
   #Out_Functional_Test.Star_Test_PLC_Functional_Test_20 := #_w1 AND #In_Functional_Test.Star_Test_PLC_Functional_Test_20;
   #Out_Functional_Test.Button_PLC_Functional_Test_20 := #_w1 AND #In_Functional_Test.Button_PLC_Functional_Test_20;
   #Out_Functional_Test.Electrical_Current_Test_Approved_PLC_Functional_Test_20 := #_w1 AND #In_Functional_Test.Electrical_Current_Test_Approved_PLC_Functional_Test_20;
   #Out_Functional_Test.Visual_Test_Approved_PLC_Functional_Test_20 := #_w1 AND #In_Functional_Test.Visual_Test_Approved_PLC_Functional_Test_20;
   IF #_w1 THEN
       #Out_Functional_Test.Electrical_Current_Read_PLC_Functional_Test_20 := #In_Functional_Test.Electrical_Current_Read_PLC_Functional_Test_20;
   END_IF;
   #Out_Functional_Test.Life_Trigger_PLC_Functional_Test_22 := #_w1 AND #In_Functional_Test.Life_Trigger_PLC_Functional_Test_22;
   #Out_Functional_Test.Star_Test_PLC_Functional_Test_22 := #_w1 AND #In_Functional_Test.Star_Test_PLC_Functional_Test_22;
   #Out_Functional_Test.Button_PLC_Functional_Test_22 := #_w1 AND #In_Functional_Test.Button_PLC_Functional_Test_22;
   #Out_Functional_Test.Electrical_Current_Test_Approved_PLC_Functional_Test_22 := #_w1 AND #In_Functional_Test.Electrical_Current_Test_Approved_PLC_Functional_Test_22;
   #Out_Functional_Test.Visual_Test_Approved_PLC_Functional_Test_22 := #_w1 AND #In_Functional_Test.Visual_Test_Approved_PLC_Functional_Test_22;
   IF #_w1 THEN
       #Out_Functional_Test.Electrical_Current_Read_PLC_Functional_Test_22 := #In_Functional_Test.Electrical_Current_Read_PLC_Functional_Test_22;
   END_IF;
   #Out_Functional_Test.Life_Trigger_PLC_Functional_Test_24 := #_w1 AND #In_Functional_Test.Life_Trigger_PLC_Functional_Test_24;
   #Out_Functional_Test.Star_Test_PLC_Functional_Test_24 := #_w1 AND #In_Functional_Test.Star_Test_PLC_Functional_Test_24;
   #Out_Functional_Test.Button_PLC_Functional_Test_24 := #_w1 AND #In_Functional_Test.Button_PLC_Functional_Test_24;
   #Out_Functional_Test.Electrical_Current_Test_Approved_PLC_Functional_Test_24 := #_w1 AND #In_Functional_Test.Electrical_Current_Test_Approved_PLC_Functional_Test_24;
   #Out_Functional_Test.Visual_Test_Approved_PLC_Functional_Test_24 := #_w1 AND #In_Functional_Test.Visual_Test_Approved_PLC_Functional_Test_24;
   IF #_w1 THEN
       #Out_Functional_Test.Electrical_Current_Read_PLC_Functional_Test_24 := #In_Functional_Test.Electrical_Current_Read_PLC_Functional_Test_24;
   END_IF;
   #Out_Functional_Test.Life_Trigger_PLC_Functional_Test_26 := #_w1 AND #In_Functional_Test.Life_Trigger_PLC_Functional_Test_26;
   #Out_Functional_Test.Star_Test_PLC_Functional_Test_26 := #_w1 AND #In_Functional_Test.Star_Test_PLC_Functional_Test_26;
   #Out_Functional_Test.Button_PLC_Functional_Test_26 := #_w1 AND #In_Functional_Test.Button_PLC_Functional_Test_26;
   #Out_Functional_Test.Electrical_Current_Test_Approved_PLC_Functional_Test_26 := #_w1 AND #In_Functional_Test.Electrical_Current_Test_Approved_PLC_Functional_Test_26;
   #Out_Functional_Test.Visual_Test_Approved_PLC_Functional_Test_26 := #_w1 AND #In_Functional_Test.Visual_Test_Approved_PLC_Functional_Test_26;
   IF #_w1 THEN
       #Out_Functional_Test.Electrical_Current_Read_PLC_Functional_Test_26 := #In_Functional_Test.Electrical_Current_Read_PLC_Functional_Test_26;
   END_IF;
   #Out_Functional_Test.Life_Trigger_PLC_Functional_Test_28 := #_w1 AND #In_Functional_Test.Life_Trigger_PLC_Functional_Test_28;
   #Out_Functional_Test.Star_Test_PLC_Functional_Test_28 := #_w1 AND #In_Functional_Test.Star_Test_PLC_Functional_Test_28;
   #Out_Functional_Test.Button_PLC_Functional_Test_28 := #_w1 AND #In_Functional_Test.Button_PLC_Functional_Test_28;
   #Out_Functional_Test.Electrical_Current_Test_Approved_PLC_Functional_Test_28 := #_w1 AND #In_Functional_Test.Electrical_Current_Test_Approved_PLC_Functional_Test_28;
   #Out_Functional_Test.Visual_Test_Approved_PLC_Functional_Test_28 := #_w1 AND #In_Functional_Test.Visual_Test_Approved_PLC_Functional_Test_28;
   IF #_w1 THEN
       #Out_Functional_Test.Electrical_Current_Read_PLC_Functional_Test_28 := #In_Functional_Test.Electrical_Current_Read_PLC_Functional_Test_28;
   END_IF;
   #Out_Functional_Test.Life_Trigger_PLC_Functional_Test_30 := #_w1 AND #In_Functional_Test.Life_Trigger_PLC_Functional_Test_30;
   #Out_Functional_Test.Star_Test_PLC_Functional_Test_30 := #_w1 AND #In_Functional_Test.Star_Test_PLC_Functional_Test_30;
   #Out_Functional_Test.Button_PLC_Functional_Test_30 := #_w1 AND #In_Functional_Test.Button_PLC_Functional_Test_30;
   #Out_Functional_Test.Electrical_Current_Test_Approved_PLC_Functional_Test_30 := #_w1 AND #In_Functional_Test.Electrical_Current_Test_Approved_PLC_Functional_Test_30;
   #Out_Functional_Test.Visual_Test_Approved_PLC_Functional_Test_30 := #_w1 AND #In_Functional_Test.Visual_Test_Approved_PLC_Functional_Test_30;
   IF #_w1 THEN
       #Out_Functional_Test.Electrical_Current_Read_PLC_Functional_Test_30 := #In_Functional_Test.Electrical_Current_Read_PLC_Functional_Test_30;
   END_IF;
END_REGION

REGION Network 7: Functional Test Station 12
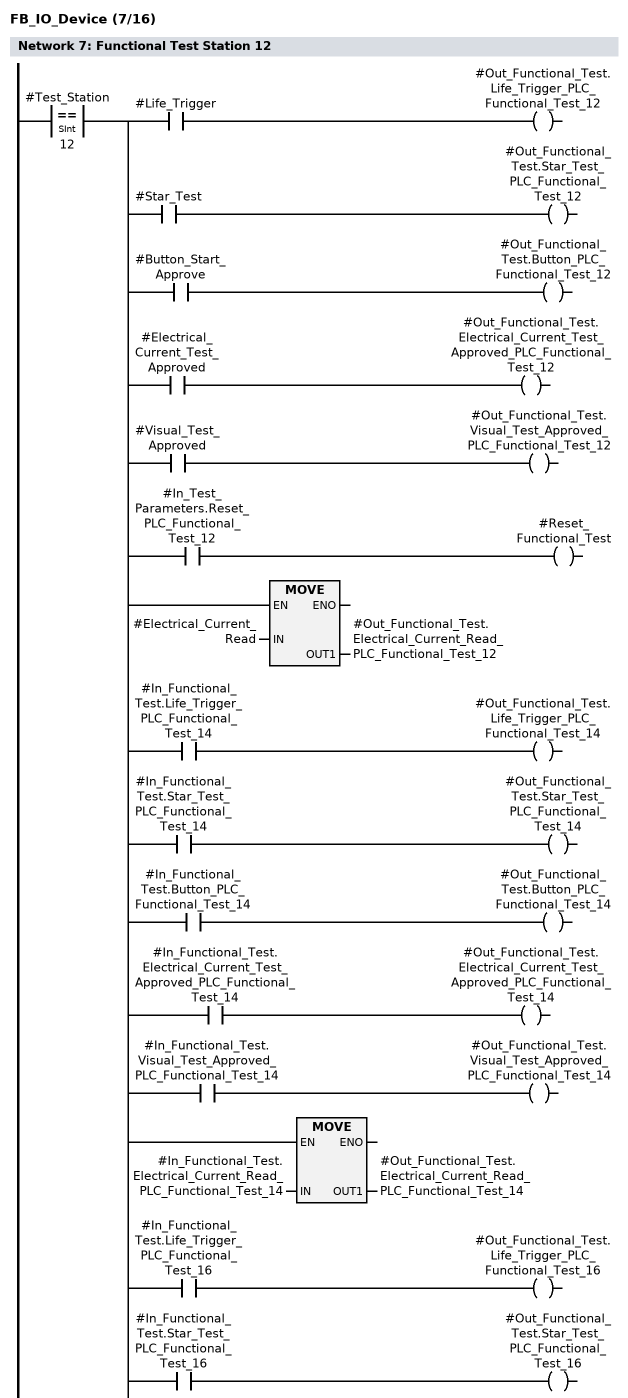
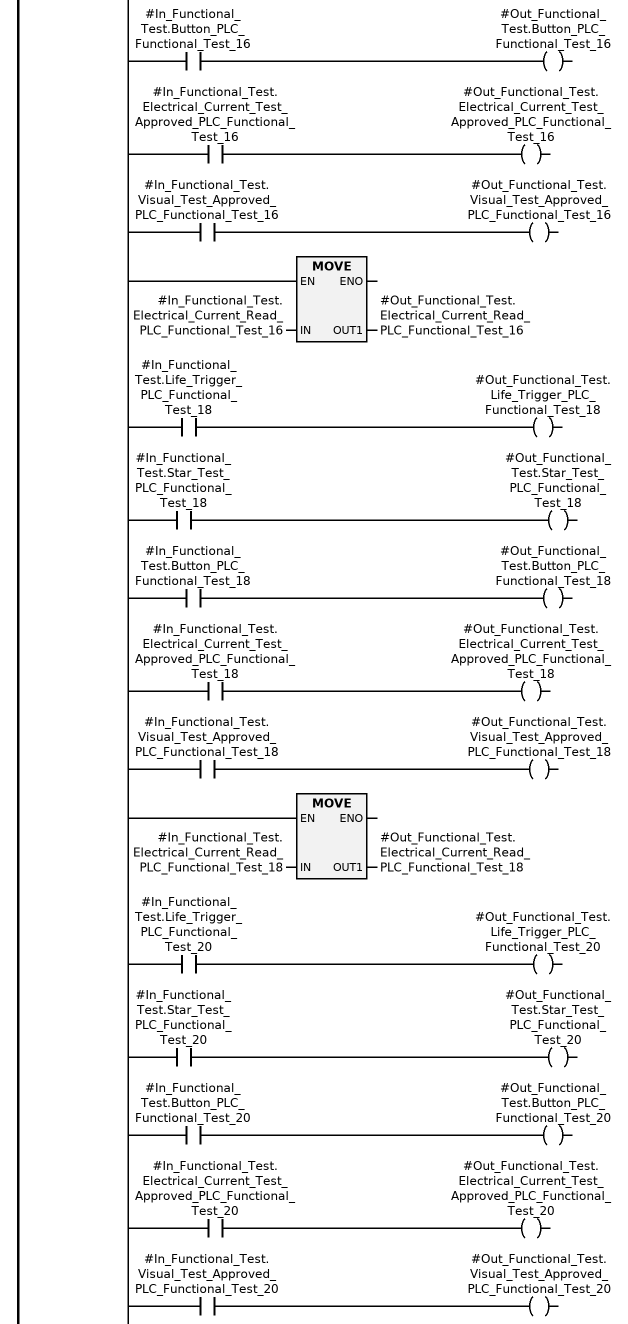
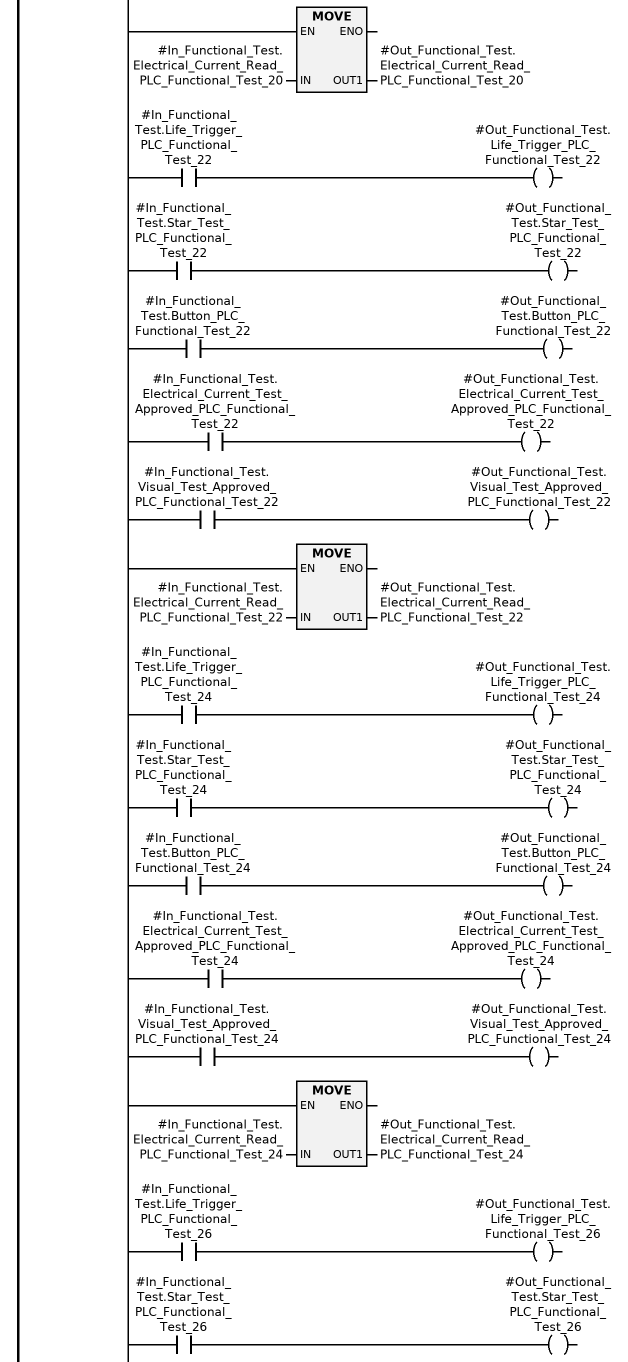
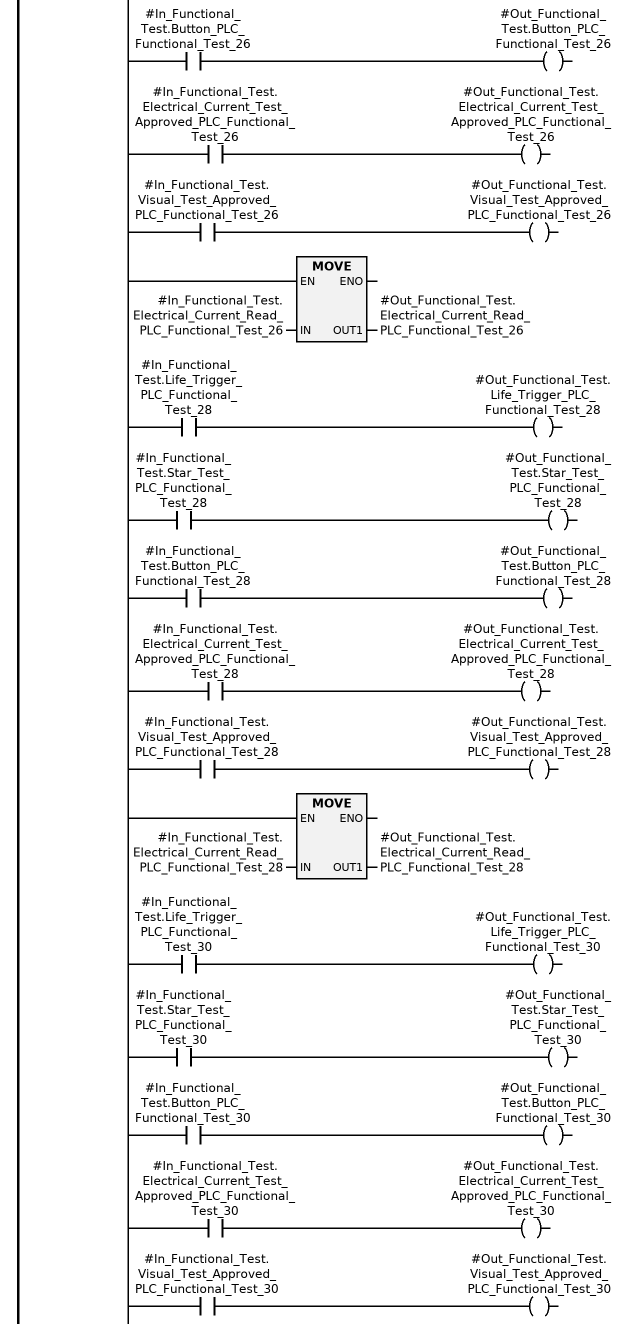
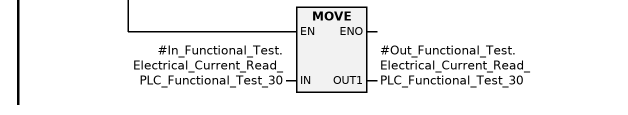
   RUNG wire#powerrail
      { S7_Templates := "SrcType := SInt" } EQ_Contact(in1 := #Test_Station, in2 := 12)
      wire#w1
      Contact( #Life_Trigger )
      Coil( #Out_Functional_Test.Life_Trigger_PLC_Functional_Test_12 )
   END_RUNG
   RUNG wire#w1
      Contact( #Star_Test )
      Coil( #Out_Functional_Test.Star_Test_PLC_Functional_Test_12 )
   END_RUNG
   RUNG wire#w1
      Contact( #Button_Start_Approve )
      Coil( #Out_Functional_Test.Button_PLC_Functional_Test_12 )
   END_RUNG
   RUNG wire#w1
      Contact( #Electrical_Current_Test_Approved )
      Coil( #Out_Functional_Test.Electrical_Current_Test_Approved_PLC_Functional_Test_12 )
   END_RUNG
   RUNG wire#w1
      Contact( #Visual_Test_Approved )
      Coil( #Out_Functional_Test.Visual_Test_Approved_PLC_Functional_Test_12 )
   END_RUNG
   RUNG wire#w1
      Contact( #In_Test_Parameters.Reset_PLC_Functional_Test_12 )
      Coil( #Reset_Functional_Test )
   END_RUNG
   RUNG wire#w1
      Move(in := #Electrical_Current_Read, out1 => #Out_Functional_Test.Electrical_Current_Read_PLC_Functional_Test_12)
   END_RUNG
   RUNG wire#w1
      Contact( #In_Functional_Test.Life_Trigger_PLC_Functional_Test_14 )
      Coil( #Out_Functional_Test.Life_Trigger_PLC_Functional_Test_14 )
   END_RUNG
   RUNG wire#w1
      Contact( #In_Functional_Test.Star_Test_PLC_Functional_Test_14 )
      Coil( #Out_Functional_Test.Star_Test_PLC_Functional_Test_14 )
   END_RUNG
   RUNG wire#w1
      Contact( #In_Functional_Test.Button_PLC_Functional_Test_14 )
      Coil( #Out_Functional_Test.Button_PLC_Functional_Test_14 )
   END_RUNG
   RUNG wire#w1
      Contact( #In_Functional_Test.Electrical_Current_Test_Approved_PLC_Functional_Test_14 )
      Coil( #Out_Functional_Test.Electrical_Current_Test_Approved_PLC_Functional_Test_14 )
   END_RUNG
   RUNG wire#w1
      Contact( #In_Functional_Test.Visual_Test_Approved_PLC_Functional_Test_14 )
      Coil( #Out_Functional_Test.Visual_Test_Approved_PLC_Functional_Test_14 )
   END_RUNG
   RUNG wire#w1
      Move(in := #In_Functional_Test.Electrical_Current_Read_PLC_Functional_Test_14, out1 => #Out_Functional_Test.Electrical_Current_Read_PLC_Functional_Test_14)
   END_RUNG
   RUNG wire#w1
      Contact( #In_Functional_Test.Life_Trigger_PLC_Functional_Test_16 )
      Coil( #Out_Functional_Test.Life_Trigger_PLC_Functional_Test_16 )
   END_RUNG
   RUNG wire#w1
      Contact( #In_Functional_Test.Star_Test_PLC_Functional_Test_16 )
      Coil( #Out_Functional_Test.Star_Test_PLC_Functional_Test_16 )
   END_RUNG
   RUNG wire#w1
      Contact( #In_Functional_Test.Button_PLC_Functional_Test_16 )
      Coil( #Out_Functional_Test.Button_PLC_Functional_Test_16 )
   END_RUNG
   RUNG wire#w1
      Contact( #In_Functional_Test.Electrical_Current_Test_Approved_PLC_Functional_Test_16 )
      Coil( #Out_Functional_Test.Electrical_Current_Test_Approved_PLC_Functional_Test_16 )
   END_RUNG
   RUNG wire#w1
      Contact( #In_Functional_Test.Visual_Test_Approved_PLC_Functional_Test_16 )
      Coil( #Out_Functional_Test.Visual_Test_Approved_PLC_Functional_Test_16 )
   END_RUNG
   RUNG wire#w1
      Move(in := #In_Functional_Test.Electrical_Current_Read_PLC_Functional_Test_16, out1 => #Out_Functional_Test.Electrical_Current_Read_PLC_Functional_Test_16)
   END_RUNG
   RUNG wire#w1
      Contact( #In_Functional_Test.Life_Trigger_PLC_Functional_Test_18 )
      Coil( #Out_Functional_Test.Life_Trigger_PLC_Functional_Test_18 )
   END_RUNG
   RUNG wire#w1
      Contact( #In_Functional_Test.Star_Test_PLC_Functional_Test_18 )
      Coil( #Out_Functional_Test.Star_Test_PLC_Functional_Test_18 )
   END_RUNG
   RUNG wire#w1
      Contact( #In_Functional_Test.Button_PLC_Functional_Test_18 )
      Coil( #Out_Functional_Test.Button_PLC_Functional_Test_18 )
   END_RUNG
   RUNG wire#w1
      Contact( #In_Functional_Test.Electrical_Current_Test_Approved_PLC_Functional_Test_18 )
      Coil( #Out_Functional_Test.Electrical_Current_Test_Approved_PLC_Functional_Test_18 )
   END_RUNG
   RUNG wire#w1
      Contact( #In_Functional_Test.Visual_Test_Approved_PLC_Functional_Test_18 )
      Coil( #Out_Functional_Test.Visual_Test_Approved_PLC_Functional_Test_18 )
   END_RUNG
   RUNG wire#w1
      Move(in := #In_Functional_Test.Electrical_Current_Read_PLC_Functional_Test_18, out1 => #Out_Functional_Test.Electrical_Current_Read_PLC_Functional_Test_18)
   END_RUNG
   RUNG wire#w1
      Contact( #In_Functional_Test.Life_Trigger_PLC_Functional_Test_20 )
      Coil( #Out_Functional_Test.Life_Trigger_PLC_Functional_Test_20 )
   END_RUNG
   RUNG wire#w1
      Contact( #In_Functional_Test.Star_Test_PLC_Functional_Test_20 )
      Coil( #Out_Functional_Test.Star_Test_PLC_Functional_Test_20 )
   END_RUNG
   RUNG wire#w1
      Contact( #In_Functional_Test.Button_PLC_Functional_Test_20 )
      Coil( #Out_Functional_Test.Button_PLC_Functional_Test_20 )
   END_RUNG
   RUNG wire#w1
      Contact( #In_Functional_Test.Electrical_Current_Test_Approved_PLC_Functional_Test_20 )
      Coil( #Out_Functional_Test.Electrical_Current_Test_Approved_PLC_Functional_Test_20 )
   END_RUNG
   RUNG wire#w1
      Contact( #In_Functional_Test.Visual_Test_Approved_PLC_Functional_Test_20 )
      Coil( #Out_Functional_Test.Visual_Test_Approved_PLC_Functional_Test_20 )
   END_RUNG
   RUNG wire#w1
      Move(in := #In_Functional_Test.Electrical_Current_Read_PLC_Functional_Test_20, out1 => #Out_Functional_Test.Electrical_Current_Read_PLC_Functional_Test_20)
   END_RUNG
   RUNG wire#w1
      Contact( #In_Functional_Test.Life_Trigger_PLC_Functional_Test_22 )
      Coil( #Out_Functional_Test.Life_Trigger_PLC_Functional_Test_22 )
   END_RUNG
   RUNG wire#w1
      Contact( #In_Functional_Test.Star_Test_PLC_Functional_Test_22 )
      Coil( #Out_Functional_Test.Star_Test_PLC_Functional_Test_22 )
   END_RUNG
   RUNG wire#w1
      Contact( #In_Functional_Test.Button_PLC_Functional_Test_22 )
      Coil( #Out_Functional_Test.Button_PLC_Functional_Test_22 )
   END_RUNG
   RUNG wire#w1
      Contact( #In_Functional_Test.Electrical_Current_Test_Approved_PLC_Functional_Test_22 )
      Coil( #Out_Functional_Test.Electrical_Current_Test_Approved_PLC_Functional_Test_22 )
   END_RUNG
   RUNG wire#w1
      Contact( #In_Functional_Test.Visual_Test_Approved_PLC_Functional_Test_22 )
      Coil( #Out_Functional_Test.Visual_Test_Approved_PLC_Functional_Test_22 )
   END_RUNG
   RUNG wire#w1
      Move(in := #In_Functional_Test.Electrical_Current_Read_PLC_Functional_Test_22, out1 => #Out_Functional_Test.Electrical_Current_Read_PLC_Functional_Test_22)
   END_RUNG
   RUNG wire#w1
      Contact( #In_Functional_Test.Life_Trigger_PLC_Functional_Test_24 )
      Coil( #Out_Functional_Test.Life_Trigger_PLC_Functional_Test_24 )
   END_RUNG
   RUNG wire#w1
      Contact( #In_Functional_Test.Star_Test_PLC_Functional_Test_24 )
      Coil( #Out_Functional_Test.Star_Test_PLC_Functional_Test_24 )
   END_RUNG
   RUNG wire#w1
      Contact( #In_Functional_Test.Button_PLC_Functional_Test_24 )
      Coil( #Out_Functional_Test.Button_PLC_Functional_Test_24 )
   END_RUNG
   RUNG wire#w1
      Contact( #In_Functional_Test.Electrical_Current_Test_Approved_PLC_Functional_Test_24 )
      Coil( #Out_Functional_Test.Electrical_Current_Test_Approved_PLC_Functional_Test_24 )
   END_RUNG
   RUNG wire#w1
      Contact( #In_Functional_Test.Visual_Test_Approved_PLC_Functional_Test_24 )
      Coil( #Out_Functional_Test.Visual_Test_Approved_PLC_Functional_Test_24 )
   END_RUNG
   RUNG wire#w1
      Move(in := #In_Functional_Test.Electrical_Current_Read_PLC_Functional_Test_24, out1 => #Out_Functional_Test.Electrical_Current_Read_PLC_Functional_Test_24)
   END_RUNG
   RUNG wire#w1
      Contact( #In_Functional_Test.Life_Trigger_PLC_Functional_Test_26 )
      Coil( #Out_Functional_Test.Life_Trigger_PLC_Functional_Test_26 )
   END_RUNG
   RUNG wire#w1
      Contact( #In_Functional_Test.Star_Test_PLC_Functional_Test_26 )
      Coil( #Out_Functional_Test.Star_Test_PLC_Functional_Test_26 )
   END_RUNG
   RUNG wire#w1
      Contact( #In_Functional_Test.Button_PLC_Functional_Test_26 )
      Coil( #Out_Functional_Test.Button_PLC_Functional_Test_26 )
   END_RUNG
   RUNG wire#w1
      Contact( #In_Functional_Test.Electrical_Current_Test_Approved_PLC_Functional_Test_26 )
      Coil( #Out_Functional_Test.Electrical_Current_Test_Approved_PLC_Functional_Test_26 )
   END_RUNG
   RUNG wire#w1
      Contact( #In_Functional_Test.Visual_Test_Approved_PLC_Functional_Test_26 )
      Coil( #Out_Functional_Test.Visual_Test_Approved_PLC_Functional_Test_26 )
   END_RUNG
   RUNG wire#w1
      Move(in := #In_Functional_Test.Electrical_Current_Read_PLC_Functional_Test_26, out1 => #Out_Functional_Test.Electrical_Current_Read_PLC_Functional_Test_26)
   END_RUNG
   RUNG wire#w1
      Contact( #In_Functional_Test.Life_Trigger_PLC_Functional_Test_28 )
      Coil( #Out_Functional_Test.Life_Trigger_PLC_Functional_Test_28 )
   END_RUNG
   RUNG wire#w1
      Contact( #In_Functional_Test.Star_Test_PLC_Functional_Test_28 )
      Coil( #Out_Functional_Test.Star_Test_PLC_Functional_Test_28 )
   END_RUNG
   RUNG wire#w1
      Contact( #In_Functional_Test.Button_PLC_Functional_Test_28 )
      Coil( #Out_Functional_Test.Button_PLC_Functional_Test_28 )
   END_RUNG
   RUNG wire#w1
      Contact( #In_Functional_Test.Electrical_Current_Test_Approved_PLC_Functional_Test_28 )
      Coil( #Out_Functional_Test.Electrical_Current_Test_Approved_PLC_Functional_Test_28 )
   END_RUNG
   RUNG wire#w1
      Contact( #In_Functional_Test.Visual_Test_Approved_PLC_Functional_Test_28 )
      Coil( #Out_Functional_Test.Visual_Test_Approved_PLC_Functional_Test_28 )
   END_RUNG
   RUNG wire#w1
      Move(in := #In_Functional_Test.Electrical_Current_Read_PLC_Functional_Test_28, out1 => #Out_Functional_Test.Electrical_Current_Read_PLC_Functional_Test_28)
   END_RUNG
   RUNG wire#w1
      Contact( #In_Functional_Test.Life_Trigger_PLC_Functional_Test_30 )
      Coil( #Out_Functional_Test.Life_Trigger_PLC_Functional_Test_30 )
   END_RUNG
   RUNG wire#w1
      Contact( #In_Functional_Test.Star_Test_PLC_Functional_Test_30 )
      Coil( #Out_Functional_Test.Star_Test_PLC_Functional_Test_30 )
   END_RUNG
   RUNG wire#w1
      Contact( #In_Functional_Test.Button_PLC_Functional_Test_30 )
      Coil( #Out_Functional_Test.Button_PLC_Functional_Test_30 )
   END_RUNG
   RUNG wire#w1
      Contact( #In_Functional_Test.Electrical_Current_Test_Approved_PLC_Functional_Test_30 )
      Coil( #Out_Functional_Test.Electrical_Current_Test_Approved_PLC_Functional_Test_30 )
   END_RUNG
   RUNG wire#w1
      Contact( #In_Functional_Test.Visual_Test_Approved_PLC_Functional_Test_30 )
      Coil( #Out_Functional_Test.Visual_Test_Approved_PLC_Functional_Test_30 )
   END_RUNG
   RUNG wire#w1
      Move(in := #In_Functional_Test.Electrical_Current_Read_PLC_Functional_Test_30, out1 => #Out_Functional_Test.Electrical_Current_Read_PLC_Functional_Test_30)
   END_RUNG
   // the same network as SCL:
   #_w1 := #Test_Station = 12;
   #Out_Functional_Test.Life_Trigger_PLC_Functional_Test_12 := #_w1 AND #Life_Trigger;
   #Out_Functional_Test.Star_Test_PLC_Functional_Test_12 := #_w1 AND #Star_Test;
   #Out_Functional_Test.Button_PLC_Functional_Test_12 := #_w1 AND #Button_Start_Approve;
   #Out_Functional_Test.Electrical_Current_Test_Approved_PLC_Functional_Test_12 := #_w1 AND #Electrical_Current_Test_Approved;
   #Out_Functional_Test.Visual_Test_Approved_PLC_Functional_Test_12 := #_w1 AND #Visual_Test_Approved;
   #Reset_Functional_Test := #_w1 AND #In_Test_Parameters.Reset_PLC_Functional_Test_12;
   IF #_w1 THEN
       #Out_Functional_Test.Electrical_Current_Read_PLC_Functional_Test_12 := #Electrical_Current_Read;
   END_IF;
   #Out_Functional_Test.Life_Trigger_PLC_Functional_Test_14 := #_w1 AND #In_Functional_Test.Life_Trigger_PLC_Functional_Test_14;
   #Out_Functional_Test.Star_Test_PLC_Functional_Test_14 := #_w1 AND #In_Functional_Test.Star_Test_PLC_Functional_Test_14;
   #Out_Functional_Test.Button_PLC_Functional_Test_14 := #_w1 AND #In_Functional_Test.Button_PLC_Functional_Test_14;
   #Out_Functional_Test.Electrical_Current_Test_Approved_PLC_Functional_Test_14 := #_w1 AND #In_Functional_Test.Electrical_Current_Test_Approved_PLC_Functional_Test_14;
   #Out_Functional_Test.Visual_Test_Approved_PLC_Functional_Test_14 := #_w1 AND #In_Functional_Test.Visual_Test_Approved_PLC_Functional_Test_14;
   IF #_w1 THEN
       #Out_Functional_Test.Electrical_Current_Read_PLC_Functional_Test_14 := #In_Functional_Test.Electrical_Current_Read_PLC_Functional_Test_14;
   END_IF;
   #Out_Functional_Test.Life_Trigger_PLC_Functional_Test_16 := #_w1 AND #In_Functional_Test.Life_Trigger_PLC_Functional_Test_16;
   #Out_Functional_Test.Star_Test_PLC_Functional_Test_16 := #_w1 AND #In_Functional_Test.Star_Test_PLC_Functional_Test_16;
   #Out_Functional_Test.Button_PLC_Functional_Test_16 := #_w1 AND #In_Functional_Test.Button_PLC_Functional_Test_16;
   #Out_Functional_Test.Electrical_Current_Test_Approved_PLC_Functional_Test_16 := #_w1 AND #In_Functional_Test.Electrical_Current_Test_Approved_PLC_Functional_Test_16;
   #Out_Functional_Test.Visual_Test_Approved_PLC_Functional_Test_16 := #_w1 AND #In_Functional_Test.Visual_Test_Approved_PLC_Functional_Test_16;
   IF #_w1 THEN
       #Out_Functional_Test.Electrical_Current_Read_PLC_Functional_Test_16 := #In_Functional_Test.Electrical_Current_Read_PLC_Functional_Test_16;
   END_IF;
   #Out_Functional_Test.Life_Trigger_PLC_Functional_Test_18 := #_w1 AND #In_Functional_Test.Life_Trigger_PLC_Functional_Test_18;
   #Out_Functional_Test.Star_Test_PLC_Functional_Test_18 := #_w1 AND #In_Functional_Test.Star_Test_PLC_Functional_Test_18;
   #Out_Functional_Test.Button_PLC_Functional_Test_18 := #_w1 AND #In_Functional_Test.Button_PLC_Functional_Test_18;
   #Out_Functional_Test.Electrical_Current_Test_Approved_PLC_Functional_Test_18 := #_w1 AND #In_Functional_Test.Electrical_Current_Test_Approved_PLC_Functional_Test_18;
   #Out_Functional_Test.Visual_Test_Approved_PLC_Functional_Test_18 := #_w1 AND #In_Functional_Test.Visual_Test_Approved_PLC_Functional_Test_18;
   IF #_w1 THEN
       #Out_Functional_Test.Electrical_Current_Read_PLC_Functional_Test_18 := #In_Functional_Test.Electrical_Current_Read_PLC_Functional_Test_18;
   END_IF;
   #Out_Functional_Test.Life_Trigger_PLC_Functional_Test_20 := #_w1 AND #In_Functional_Test.Life_Trigger_PLC_Functional_Test_20;
   #Out_Functional_Test.Star_Test_PLC_Functional_Test_20 := #_w1 AND #In_Functional_Test.Star_Test_PLC_Functional_Test_20;
   #Out_Functional_Test.Button_PLC_Functional_Test_20 := #_w1 AND #In_Functional_Test.Button_PLC_Functional_Test_20;
   #Out_Functional_Test.Electrical_Current_Test_Approved_PLC_Functional_Test_20 := #_w1 AND #In_Functional_Test.Electrical_Current_Test_Approved_PLC_Functional_Test_20;
   #Out_Functional_Test.Visual_Test_Approved_PLC_Functional_Test_20 := #_w1 AND #In_Functional_Test.Visual_Test_Approved_PLC_Functional_Test_20;
   IF #_w1 THEN
       #Out_Functional_Test.Electrical_Current_Read_PLC_Functional_Test_20 := #In_Functional_Test.Electrical_Current_Read_PLC_Functional_Test_20;
   END_IF;
   #Out_Functional_Test.Life_Trigger_PLC_Functional_Test_22 := #_w1 AND #In_Functional_Test.Life_Trigger_PLC_Functional_Test_22;
   #Out_Functional_Test.Star_Test_PLC_Functional_Test_22 := #_w1 AND #In_Functional_Test.Star_Test_PLC_Functional_Test_22;
   #Out_Functional_Test.Button_PLC_Functional_Test_22 := #_w1 AND #In_Functional_Test.Button_PLC_Functional_Test_22;
   #Out_Functional_Test.Electrical_Current_Test_Approved_PLC_Functional_Test_22 := #_w1 AND #In_Functional_Test.Electrical_Current_Test_Approved_PLC_Functional_Test_22;
   #Out_Functional_Test.Visual_Test_Approved_PLC_Functional_Test_22 := #_w1 AND #In_Functional_Test.Visual_Test_Approved_PLC_Functional_Test_22;
   IF #_w1 THEN
       #Out_Functional_Test.Electrical_Current_Read_PLC_Functional_Test_22 := #In_Functional_Test.Electrical_Current_Read_PLC_Functional_Test_22;
   END_IF;
   #Out_Functional_Test.Life_Trigger_PLC_Functional_Test_24 := #_w1 AND #In_Functional_Test.Life_Trigger_PLC_Functional_Test_24;
   #Out_Functional_Test.Star_Test_PLC_Functional_Test_24 := #_w1 AND #In_Functional_Test.Star_Test_PLC_Functional_Test_24;
   #Out_Functional_Test.Button_PLC_Functional_Test_24 := #_w1 AND #In_Functional_Test.Button_PLC_Functional_Test_24;
   #Out_Functional_Test.Electrical_Current_Test_Approved_PLC_Functional_Test_24 := #_w1 AND #In_Functional_Test.Electrical_Current_Test_Approved_PLC_Functional_Test_24;
   #Out_Functional_Test.Visual_Test_Approved_PLC_Functional_Test_24 := #_w1 AND #In_Functional_Test.Visual_Test_Approved_PLC_Functional_Test_24;
   IF #_w1 THEN
       #Out_Functional_Test.Electrical_Current_Read_PLC_Functional_Test_24 := #In_Functional_Test.Electrical_Current_Read_PLC_Functional_Test_24;
   END_IF;
   #Out_Functional_Test.Life_Trigger_PLC_Functional_Test_26 := #_w1 AND #In_Functional_Test.Life_Trigger_PLC_Functional_Test_26;
   #Out_Functional_Test.Star_Test_PLC_Functional_Test_26 := #_w1 AND #In_Functional_Test.Star_Test_PLC_Functional_Test_26;
   #Out_Functional_Test.Button_PLC_Functional_Test_26 := #_w1 AND #In_Functional_Test.Button_PLC_Functional_Test_26;
   #Out_Functional_Test.Electrical_Current_Test_Approved_PLC_Functional_Test_26 := #_w1 AND #In_Functional_Test.Electrical_Current_Test_Approved_PLC_Functional_Test_26;
   #Out_Functional_Test.Visual_Test_Approved_PLC_Functional_Test_26 := #_w1 AND #In_Functional_Test.Visual_Test_Approved_PLC_Functional_Test_26;
   IF #_w1 THEN
       #Out_Functional_Test.Electrical_Current_Read_PLC_Functional_Test_26 := #In_Functional_Test.Electrical_Current_Read_PLC_Functional_Test_26;
   END_IF;
   #Out_Functional_Test.Life_Trigger_PLC_Functional_Test_28 := #_w1 AND #In_Functional_Test.Life_Trigger_PLC_Functional_Test_28;
   #Out_Functional_Test.Star_Test_PLC_Functional_Test_28 := #_w1 AND #In_Functional_Test.Star_Test_PLC_Functional_Test_28;
   #Out_Functional_Test.Button_PLC_Functional_Test_28 := #_w1 AND #In_Functional_Test.Button_PLC_Functional_Test_28;
   #Out_Functional_Test.Electrical_Current_Test_Approved_PLC_Functional_Test_28 := #_w1 AND #In_Functional_Test.Electrical_Current_Test_Approved_PLC_Functional_Test_28;
   #Out_Functional_Test.Visual_Test_Approved_PLC_Functional_Test_28 := #_w1 AND #In_Functional_Test.Visual_Test_Approved_PLC_Functional_Test_28;
   IF #_w1 THEN
       #Out_Functional_Test.Electrical_Current_Read_PLC_Functional_Test_28 := #In_Functional_Test.Electrical_Current_Read_PLC_Functional_Test_28;
   END_IF;
   #Out_Functional_Test.Life_Trigger_PLC_Functional_Test_30 := #_w1 AND #In_Functional_Test.Life_Trigger_PLC_Functional_Test_30;
   #Out_Functional_Test.Star_Test_PLC_Functional_Test_30 := #_w1 AND #In_Functional_Test.Star_Test_PLC_Functional_Test_30;
   #Out_Functional_Test.Button_PLC_Functional_Test_30 := #_w1 AND #In_Functional_Test.Button_PLC_Functional_Test_30;
   #Out_Functional_Test.Electrical_Current_Test_Approved_PLC_Functional_Test_30 := #_w1 AND #In_Functional_Test.Electrical_Current_Test_Approved_PLC_Functional_Test_30;
   #Out_Functional_Test.Visual_Test_Approved_PLC_Functional_Test_30 := #_w1 AND #In_Functional_Test.Visual_Test_Approved_PLC_Functional_Test_30;
   IF #_w1 THEN
       #Out_Functional_Test.Electrical_Current_Read_PLC_Functional_Test_30 := #In_Functional_Test.Electrical_Current_Read_PLC_Functional_Test_30;
   END_IF;
END_REGION

REGION Network 8: Functional Test Station 14
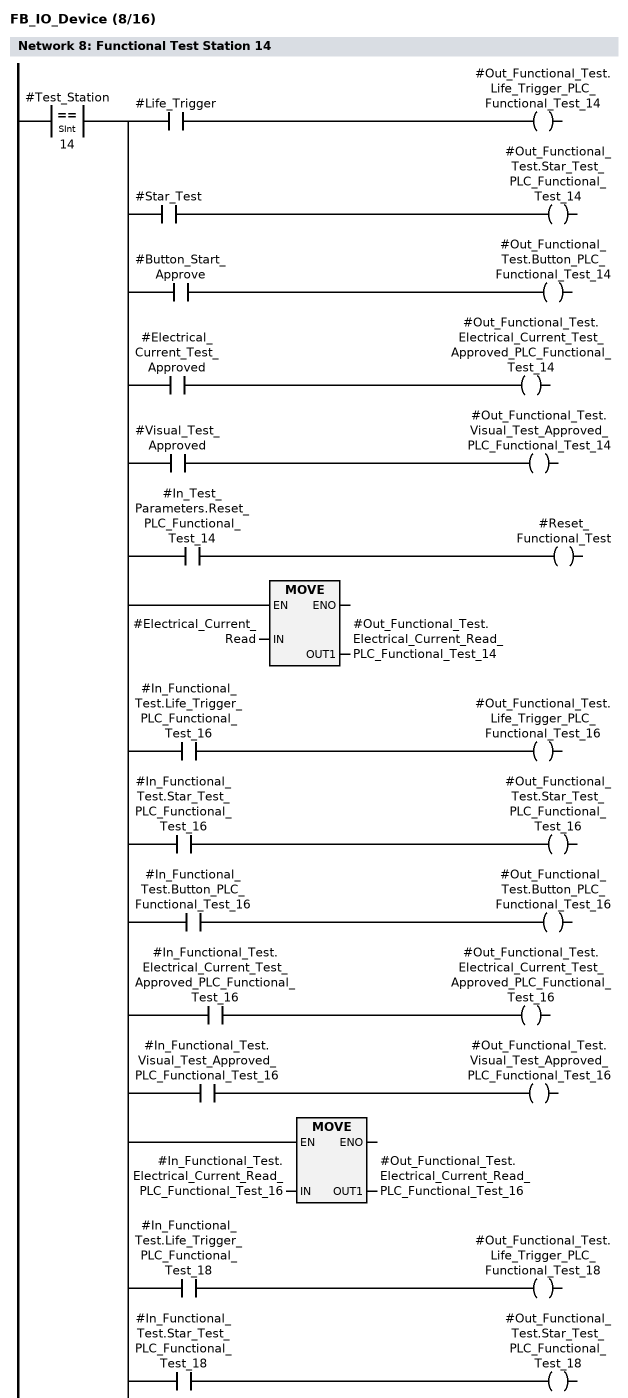
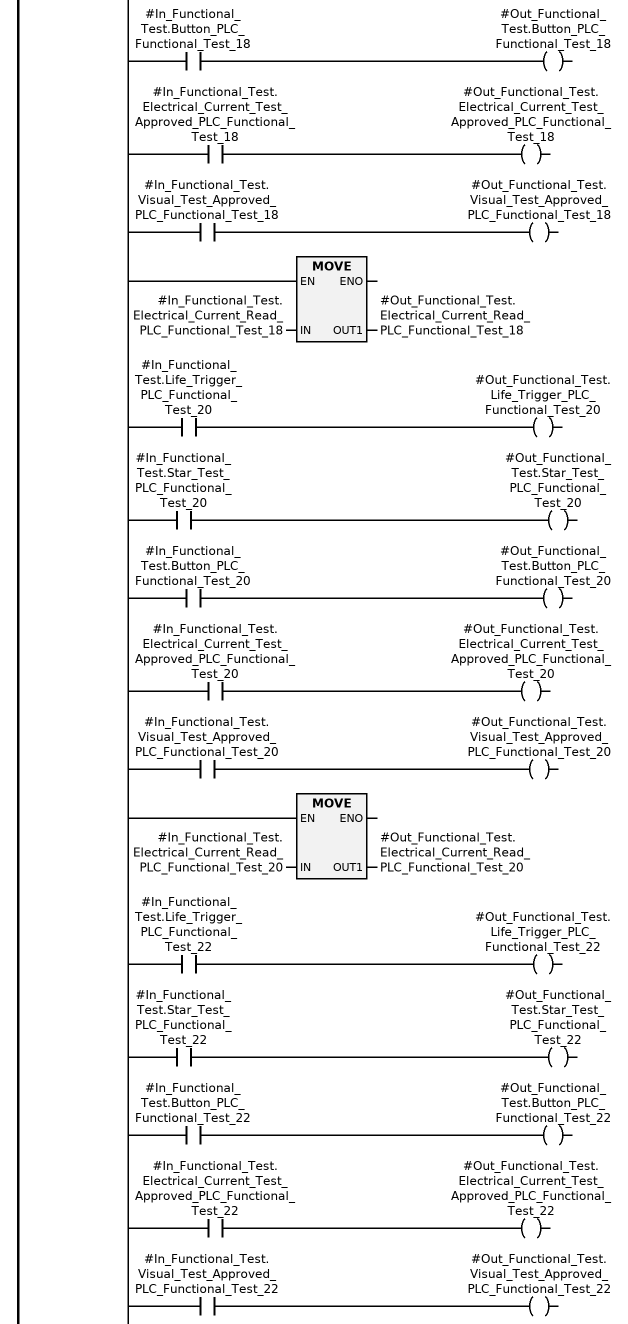
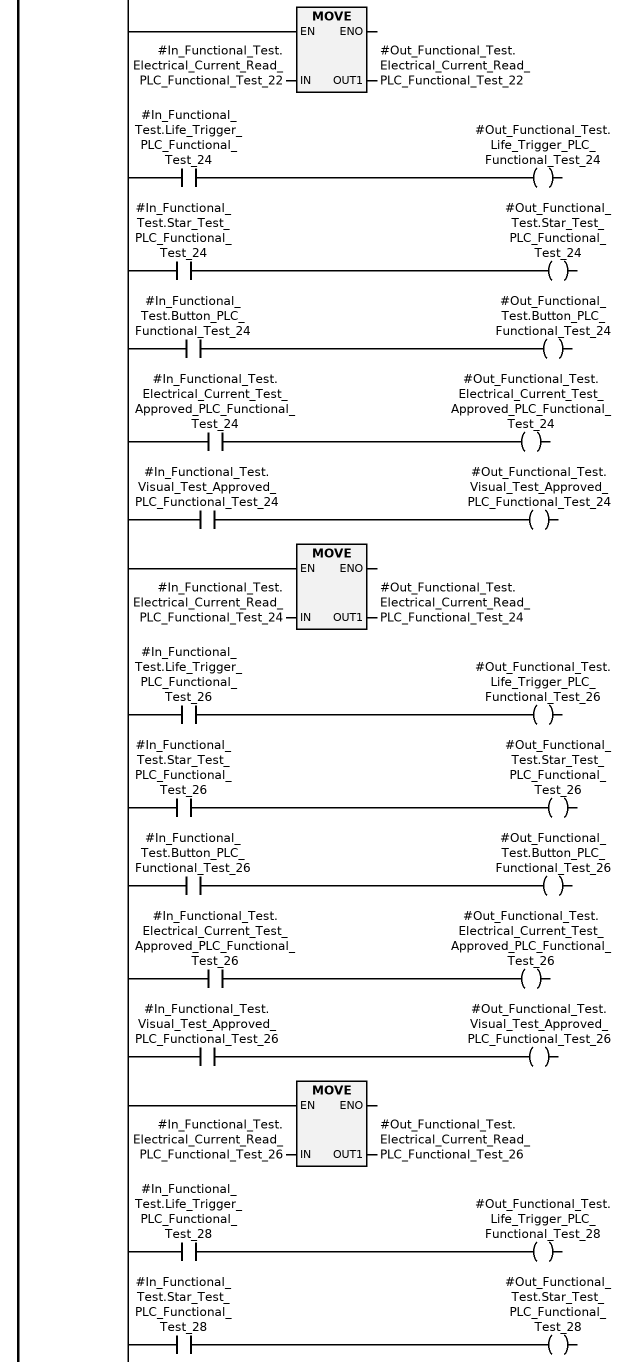
